LIN {X 0.130,Y -388.689,Z 418.603,A 0.000,B 0.000,C 90.000,E1 108.489} C_DIS
LIN {X -0.134,Y -405.495,Z 418.590,A 0.000,B 0.000,C 90.000,E1 106.260} C_DIS
LIN {X 0.180,Y -423.948,Z 418.578,A 0.000,B 0.000,C 90.000,E1 104.008} C_DIS
LIN {X -0.236,Y -443.839,Z 418.566,A 0.000,B 0.000,C 90.000,E1 101.951} C_DIS
LIN {X 0.157,Y -464.340,Z 418.555,A 0.000,B 0.000,C 90.000,E1 99.962} C_DIS
LIN {X -0.148,Y -485.345,Z 418.546,A 0.000,B 0.000,C 90.000,E1 98.219} C_DIS
LIN {X -0.012,Y -487.672,Z 418.544,A 0.000,B 0.000,C 90.000,E1 97.992} C_DIS
LIN {X 0.194,Y -489.436,Z 418.543,A 0.000,B 0.000,C 90.000,E1 97.757} C_DIS
LIN {X 0.023,Y -491.019,Z 418.542,A 0.000,B 0.000,C 90.000,E1 97.530} C_DIS
LIN {X -0.083,Y -492.202,Z 418.540,A 0.000,B 0.000,C 90.000,E1 97.296} C_DIS
LIN {X 0.146,Y -493.628,Z 418.538,A 0.000,B 0.000,C 90.000,E1 96.777} C_DIS
LIN {X -0.107,Y -494.007,Z 418.535,A 0.000,B 0.000,C 90.000,E1 96.315} C_DIS
LIN {X 0.138,Y -493.395,Z 418.532,A 0.000,B 0.000,C 90.000,E1 95.796} C_DIS
LIN {X -0.107,Y -491.696,Z 418.530,A 0.000,B 0.000,C 90.000,E1 95.334} C_DIS
LIN {X 0.236,Y -490.338,Z 418.528,A 0.000,B 0.000,C 90.000,E1 95.049} C_DIS
LIN {X -0.171,Y -484.764,Z 418.524,A 0.000,B 0.000,C 90.000,E1 94.359} C_DIS
LIN {X -0.157,Y -472.832,Z 418.516,A 0.000,B 0.000,C 90.000,E1 92.865} C_DIS
LIN {X -0.097,Y -455.462,Z 418.503,A 0.000,B 0.000,C 90.000,E1 90.573} C_DIS
LIN {X 0.061,Y -434.620,Z 418.486,A 0.000,B 0.000,C 90.000,E1 87.421} C_DIS
LIN {X 0.132,Y -413.786,Z 418.466,A 0.000,B 0.000,C 90.000,E1 83.913} C_DIS
LIN {X 0.008,Y -401.504,Z 418.454,A 0.000,B 0.000,C 90.000,E1 81.724} C_DIS
LIN {X 0.096,Y -390.851,Z 418.443,A 0.000,B 0.000,C 90.000,E1 79.746} C_DIS
LIN {X 0.073,Y -378.899,Z 418.430,A 0.000,B 0.000,C 90.000,E1 77.465} C_DIS
LIN {X -0.069,Y -365.997,Z 418.416,A 0.000,B 0.000,C 90.000,E1 74.866} C_DIS
LIN {X -0.041,Y -350.988,Z 418.398,A 0.000,B 0.000,C 90.000,E1 71.583} C_DIS
LIN {X -0.070,Y -338.219,Z 418.381,A 0.000,B 0.000,C 90.000,E1 68.539} C_DIS
LIN {X -0.050,Y -328.301,Z 418.367,A 0.000,B 0.000,C 90.000,E1 66.049} C_DIS
LIN {X 0.061,Y -319.808,Z 418.355,A 0.000,B 0.000,C 90.000,E1 63.819} C_DIS
LIN {X 0.144,Y -308.074,Z 418.337,A 0.000,B 0.000,C 90.000,E1 60.589} C_DIS
LIN {X 0.043,Y -297.005,Z 418.319,A 0.000,B 0.000,C 90.000,E1 57.327} C_DIS
LIN {X 0.032,Y -286.983,Z 418.300,A 0.000,B 0.000,C 90.000,E1 53.989} C_DIS
LIN {X 0.145,Y -279.385,Z 418.285,A 0.000,B 0.000,C 90.000,E1 51.251} C_DIS
LIN {X 0.000,Y -273.756,Z 418.273,A 0.000,B 0.000,C 90.000,E1 49.218} C_DIS
LIN {X -0.063,Y -267.896,Z 418.262,A 0.000,B 0.000,C 90.000,E1 47.148} C_DIS
LIN {X 0.124,Y -261.832,Z 418.250,A 0.000,B 0.000,C 90.000,E1 45.000} C_DIS
LIN {X 0.005,Y -255.633,Z 418.238,A 0.000,B 0.000,C 90.000,E1 42.894} C_DIS
LIN {X 0.002,Y -247.147,Z 418.222,A 0.000,B 0.000,C 90.000,E1 40.011} C_DIS
LIN {X -0.019,Y -236.856,Z 418.202,A 0.000,B 0.000,C 90.000,E1 36.343} C_DIS
LIN {X -0.108,Y -229.315,Z 418.185,A 0.000,B 0.000,C 90.000,E1 33.372} C_DIS
LIN {X -0.114,Y -222.425,Z 418.168,A 0.000,B 0.000,C 90.000,E1 30.335} C_DIS
LIN {X 0.062,Y -216.232,Z 418.151,A 0.000,B 0.000,C 90.000,E1 27.206} C_DIS
LIN {X -0.079,Y -209.441,Z 418.130,A 0.000,B 0.000,C 90.000,E1 23.334} C_DIS
LIN {X 0.087,Y -203.617,Z 418.107,A 0.000,B 0.000,C 90.000,E1 19.322} C_DIS
LIN {X 0.059,Y -198.758,Z 418.085,A 0.000,B 0.000,C 90.000,E1 15.315} C_DIS
LIN {X -0.095,Y -194.212,Z 418.058,A 0.000,B 0.000,C 90.000,E1 10.489} C_DIS
LIN {X -0.079,Y -191.040,Z 418.031,A 0.000,B 0.000,C 90.000,E1 5.568} C_DIS
LIN {X 0.073,Y -189.334,Z 417.993,A 0.000,B 0.000,C 90.000,E1 358.682} C_DIS
LIN {X -0.003,Y -191.373,Z 417.947,A 0.000,B 0.000,C 90.000,E1 350.443} C_DIS
LIN {X -0.026,Y -194.437,Z 417.919,A 0.000,B 0.000,C 90.000,E1 345.519} C_DIS
LIN {X -0.091,Y -198.077,Z 417.897,A 0.000,B 0.000,C 90.000,E1 341.456} C_DIS
LIN {X 0.089,Y -202.701,Z 417.874,A 0.000,B 0.000,C 90.000,E1 337.358} C_DIS
LIN {X -0.017,Y -208.427,Z 417.852,A 0.000,B 0.000,C 90.000,E1 333.384} C_DIS
LIN {X 0.026,Y -213.606,Z 417.835,A 0.000,B 0.000,C 90.000,E1 330.205} C_DIS
LIN {X 0.038,Y -220.600,Z 417.813,A 0.000,B 0.000,C 90.000,E1 326.294} C_DIS
LIN {X -0.092,Y -228.187,Z 417.791,A 0.000,B 0.000,C 90.000,E1 322.477} C_DIS
LIN {X -0.103,Y -236.777,Z 417.770,A 0.000,B 0.000,C 90.000,E1 318.690} C_DIS
LIN {X -0.037,Y -245.598,Z 417.752,A 0.000,B 0.000,C 90.000,E1 315.324} C_DIS
LIN {X 0.115,Y -254.400,Z 417.736,A 0.000,B 0.000,C 90.000,E1 312.366} C_DIS
LIN {X -0.143,Y -265.533,Z 417.718,A 0.000,B 0.000,C 90.000,E1 309.197} C_DIS
LIN {X 0.003,Y -277.655,Z 417.700,A 0.000,B 0.000,C 90.000,E1 306.011} C_DIS
LIN {X -0.128,Y -289.063,Z 417.685,A 0.000,B 0.000,C 90.000,E1 303.293} C_DIS
LIN {X -0.018,Y -303.956,Z 417.666,A 0.000,B 0.000,C 90.000,E1 299.922} C_DIS
LIN {X -0.031,Y -320.508,Z 417.648,A 0.000,B 0.000,C 90.000,E1 296.668} C_DIS
LIN {X -0.034,Y -335.095,Z 417.634,A 0.000,B 0.000,C 90.000,E1 294.131} C_DIS
LIN {X -0.001,Y -355.906,Z 417.617,A 0.000,B 0.000,C 90.000,E1 291.046} C_DIS
LIN {X 0.014,Y -376.407,Z 417.602,A 0.000,B 0.000,C 90.000,E1 288.362} C_DIS
LIN {X 0.077,Y -388.412,Z 417.594,A 0.000,B 0.000,C 90.000,E1 286.913} C_DIS
LIN {X 0.102,Y -403.817,Z 417.585,A 0.000,B 0.000,C 90.000,E1 285.245} C_DIS
LIN {X -0.137,Y -422.217,Z 417.575,A 0.000,B 0.000,C 90.000,E1 283.467} C_DIS
LIN {X 0.197,Y -432.492,Z 417.569,A 0.000,B 0.000,C 90.000,E1 282.411} C_DIS
LIN {X 0.001,Y -442.349,Z 417.563,A 0.000,B 0.000,C 90.000,E1 281.422} C_DIS
LIN {X -0.183,Y -449.356,Z 417.559,A 0.000,B 0.000,C 90.000,E1 280.658} C_DIS
LIN {X 0.023,Y -455.862,Z 417.555,A 0.000,B 0.000,C 90.000,E1 279.849} C_DIS
LIN {X 0.128,Y -463.718,Z 417.549,A 0.000,B 0.000,C 90.000,E1 278.803} C_DIS
LIN {X -0.141,Y -470.785,Z 417.543,A 0.000,B 0.000,C 90.000,E1 277.814} C_DIS
LIN {X -0.252,Y -475.616,Z 417.539,A 0.000,B 0.000,C 90.000,E1 277.068} C_DIS
LIN {X 0.210,Y -480.072,Z 417.535,A 0.000,B 0.000,C 90.000,E1 276.258} C_DIS
LIN {X 0.190,Y -484.015,Z 417.531,A 0.000,B 0.000,C 90.000,E1 275.511} C_DIS
LIN {X 0.243,Y -487.204,Z 417.527,A 0.000,B 0.000,C 90.000,E1 274.759} C_DIS
LIN {X -0.084,Y -488.885,Z 417.524,A 0.000,B 0.000,C 90.000,E1 274.302} C_DIS
LIN {X 0.119,Y -490.191,Z 417.521,A 0.000,B 0.000,C 90.000,E1 273.784} C_DIS
LIN {X -0.188,Y -491.163,Z 417.518,A 0.000,B 0.000,C 90.000,E1 273.326} C_DIS
LIN {X 0.030,Y -491.852,Z 417.516,A 0.000,B 0.000,C 90.000,E1 272.808} C_DIS
LIN {X 0.229,Y -492.166,Z 417.513,A 0.000,B 0.000,C 90.000,E1 272.293} C_DIS
LIN {X -0.058,Y -492.088,Z 417.510,A 0.000,B 0.000,C 90.000,E1 271.835} C_DIS
LIN {X 0.164,Y -491.562,Z 417.507,A 0.000,B 0.000,C 90.000,E1 271.318} C_DIS
LIN {X -0.120,Y -490.645,Z 417.505,A 0.000,B 0.000,C 90.000,E1 270.859} C_DIS
LIN {X 0.084,Y -489.178,Z 417.502,A 0.000,B 0.000,C 90.000,E1 270.344} C_DIS
LIN {X -0.205,Y -487.193,Z 417.499,A 0.000,B 0.000,C 90.000,E1 269.885} C_DIS
LIN {X -0.014,Y -484.575,Z 417.496,A 0.000,B 0.000,C 90.000,E1 269.370} C_DIS
LIN {X 0.154,Y -481.265,Z 417.494,A 0.000,B 0.000,C 90.000,E1 268.854} C_DIS
LIN {X -0.174,Y -477.014,Z 417.491,A 0.000,B 0.000,C 90.000,E1 268.396} C_DIS
LIN {X -0.030,Y -471.634,Z 417.488,A 0.000,B 0.000,C 90.000,E1 267.879} C_DIS
LIN {X -0.022,Y -468.790,Z 417.487,A 0.000,B 0.000,C 90.000,E1 267.650} C_DIS
LIN {X -0.013,Y -465.536,Z 417.486,A 0.000,B 0.000,C 90.000,E1 267.421} C_DIS
LIN {X -0.198,Y -462.346,Z 417.485,A 0.000,B 0.000,C 90.000,E1 267.249} C_DIS
LIN {X -0.238,Y -455.324,Z 417.483,A 0.000,B 0.000,C 90.000,E1 266.906} C_DIS
LIN {X -0.153,Y -448.247,Z 417.481,A 0.000,B 0.000,C 90.000,E1 266.617} C_DIS
LIN {X -0.141,Y -440.917,Z 417.480,A 0.000,B 0.000,C 90.000,E1 266.388} C_DIS
LIN {X -0.216,Y -433.025,Z 417.479,A 0.000,B 0.000,C 90.000,E1 266.216} C_DIS
LIN {X 0.047,Y -424.526,Z 417.478,A 0.000,B 0.000,C 90.000,E1 266.045} C_DIS
LIN {X 0.186,Y -412.102,Z 417.478,A 0.000,B 0.000,C 90.000,E1 265.931} C_DIS
LIN {X 0.148,Y -409.362,Z 417.477,A 0.000,B 0.000,C 90.000,E1 265.927} C_DIS
LIN {X 0.036,Y -180.917,Z 417.477,A 0.000,B 0.000,C 90.000,E1 265.927} C_DIS
LIN {X 0.040,Y -180.838,Z 417.472,A 0.000,B 0.000,C 90.000,E1 264.894} C_DIS
LIN {X -0.063,Y -178.878,Z 417.443,A 0.000,B 0.000,C 90.000,E1 259.690} C_DIS
LIN {X 0.013,Y -175.921,Z 417.414,A 0.000,B 0.000,C 90.000,E1 254.574} C_DIS
LIN {X -0.098,Y -174.618,Z 417.405,A 0.000,B 0.000,C 90.000,E1 252.906} C_DIS
LIN {X -0.005,Y -171.599,Z 417.381,A 0.000,B 0.000,C 90.000,E1 248.592} C_DIS
LIN {X -0.016,Y -167.821,Z 417.357,A 0.000,B 0.000,C 90.000,E1 244.280} C_DIS
LIN {X 0.001,Y -166.546,Z 417.347,A 0.000,B 0.000,C 90.000,E1 242.538} C_DIS
LIN {X -0.089,Y -162.542,Z 417.323,A 0.000,B 0.000,C 90.000,E1 238.201} C_DIS
LIN {X -0.028,Y -161.219,Z 417.313,A 0.000,B 0.000,C 90.000,E1 236.421} C_DIS
LIN {X 0.007,Y -157.226,Z 417.289,A 0.000,B 0.000,C 90.000,E1 231.984} C_DIS
LIN {X 0.031,Y -155.951,Z 417.279,A 0.000,B 0.000,C 90.000,E1 230.194} C_DIS
LIN {X -0.011,Y -152.205,Z 417.254,A 0.000,B 0.000,C 90.000,E1 225.729} C_DIS
LIN {X 0.011,Y -150.450,Z 417.239,A 0.000,B 0.000,C 90.000,E1 223.014} C_DIS
LIN {X 0.037,Y -147.176,Z 417.214,A 0.000,B 0.000,C 90.000,E1 218.463} C_DIS
LIN {X 0.004,Y -145.193,Z 417.193,A 0.000,B 0.000,C 90.000,E1 214.818} C_DIS
LIN {X 0.039,Y -142.333,Z 417.163,A 0.000,B 0.000,C 90.000,E1 209.283} C_DIS
LIN {X -0.032,Y -141.722,Z 417.152,A 0.000,B 0.000,C 90.000,E1 207.462} C_DIS
LIN {X -0.049,Y -139.478,Z 417.116,A 0.000,B 0.000,C 90.000,E1 200.972} C_DIS
LIN {X -0.061,Y -138.976,Z 417.101,A 0.000,B 0.000,C 90.000,E1 198.181} C_DIS
LIN {X 0.061,Y -138.331,Z 417.054,A 0.000,B 0.000,C 90.000,E1 189.726} C_DIS
LIN {X 0.064,Y -139.432,Z 417.007,A 0.000,B 0.000,C 90.000,E1 181.318} C_DIS
LIN {X 0.004,Y -140.959,Z 416.976,A 0.000,B 0.000,C 90.000,E1 175.755} C_DIS
LIN {X -0.046,Y -142.715,Z 416.956,A 0.000,B 0.000,C 90.000,E1 172.064} C_DIS
LIN {X 0.054,Y -145.094,Z 416.930,A 0.000,B 0.000,C 90.000,E1 167.409} C_DIS
LIN {X 0.049,Y -147.718,Z 416.910,A 0.000,B 0.000,C 90.000,E1 163.740} C_DIS
LIN {X -0.010,Y -150.375,Z 416.889,A 0.000,B 0.000,C 90.000,E1 160.115} C_DIS
LIN {X 0.008,Y -153.805,Z 416.869,A 0.000,B 0.000,C 90.000,E1 156.485} C_DIS
LIN {X 0.068,Y -157.216,Z 416.849,A 0.000,B 0.000,C 90.000,E1 152.871} C_DIS
LIN {X 0.008,Y -161.381,Z 416.830,A 0.000,B 0.000,C 90.000,E1 149.331} C_DIS
LIN {X 0.020,Y -165.583,Z 416.810,A 0.000,B 0.000,C 90.000,E1 145.801} C_DIS
LIN {X 0.006,Y -170.506,Z 416.791,A 0.000,B 0.000,C 90.000,E1 142.316} C_DIS
LIN {X 0.050,Y -175.385,Z 416.771,A 0.000,B 0.000,C 90.000,E1 138.852} C_DIS
LIN {X -0.087,Y -181.009,Z 416.753,A 0.000,B 0.000,C 90.000,E1 135.486} C_DIS
LIN {X 0.037,Y -186.439,Z 416.734,A 0.000,B 0.000,C 90.000,E1 132.081} C_DIS
LIN {X 0.106,Y -191.064,Z 416.720,A 0.000,B 0.000,C 90.000,E1 129.564} C_DIS
LIN {X -0.035,Y -196.732,Z 416.702,A 0.000,B 0.000,C 90.000,E1 126.377} C_DIS
LIN {X -0.087,Y -294.757,Z 416.702,A 0.000,B 0.000,C 90.000,E1 126.377} C_DIS
LIN {X 0.042,Y -297.998,Z 416.702,A 0.000,B 0.000,C 90.000,E1 126.297} C_DIS
LIN {X 0.063,Y -300.668,Z 416.701,A 0.000,B 0.000,C 90.000,E1 126.171} C_DIS
LIN {X 0.071,Y -304.249,Z 416.699,A 0.000,B 0.000,C 90.000,E1 125.884} C_DIS
LIN {X -0.057,Y -307.884,Z 416.697,A 0.000,B 0.000,C 90.000,E1 125.438} C_DIS
LIN {X -0.031,Y -309.677,Z 416.695,A 0.000,B 0.000,C 90.000,E1 125.105} C_DIS
LIN {X -0.004,Y -311.083,Z 416.693,A 0.000,B 0.000,C 90.000,E1 124.771} C_DIS
LIN {X 0.092,Y -323.167,Z 416.673,A 0.000,B 0.000,C 90.000,E1 121.209} C_DIS
LIN {X 0.136,Y -334.446,Z 416.658,A 0.000,B 0.000,C 90.000,E1 118.359} C_DIS
LIN {X 0.024,Y -347.149,Z 416.642,A 0.000,B 0.000,C 90.000,E1 115.591} C_DIS
LIN {X 0.094,Y -359.734,Z 416.629,A 0.000,B 0.000,C 90.000,E1 113.153} C_DIS
LIN {X 0.010,Y -373.629,Z 416.616,A 0.000,B 0.000,C 90.000,E1 110.791} C_DIS
LIN {X -0.133,Y -388.936,Z 416.603,A 0.000,B 0.000,C 90.000,E1 108.489} C_DIS
LIN {X -0.013,Y -405.767,Z 416.590,A 0.000,B 0.000,C 90.000,E1 106.205} C_DIS
LIN {X -0.093,Y -424.249,Z 416.578,A 0.000,B 0.000,C 90.000,E1 104.008} C_DIS
LIN {X 0.024,Y -444.153,Z 416.566,A 0.000,B 0.000,C 90.000,E1 101.883} C_DIS
LIN {X -0.099,Y -464.664,Z 416.555,A 0.000,B 0.000,C 90.000,E1 99.962} C_DIS
LIN {X 0.086,Y -485.676,Z 416.545,A 0.000,B 0.000,C 90.000,E1 98.163} C_DIS
LIN {X 0.207,Y -487.985,Z 416.544,A 0.000,B 0.000,C 90.000,E1 97.936} C_DIS
LIN {X 0.231,Y -489.872,Z 416.543,A 0.000,B 0.000,C 90.000,E1 97.701} C_DIS
LIN {X 0.190,Y -491.309,Z 416.542,A 0.000,B 0.000,C 90.000,E1 97.473} C_DIS
LIN {X -0.013,Y -493.295,Z 416.539,A 0.000,B 0.000,C 90.000,E1 97.004} C_DIS
LIN {X 0.217,Y -494.139,Z 416.536,A 0.000,B 0.000,C 90.000,E1 96.486} C_DIS
LIN {X -0.084,Y -493.986,Z 416.533,A 0.000,B 0.000,C 90.000,E1 96.030} C_DIS
LIN {X 0.166,Y -492.812,Z 416.531,A 0.000,B 0.000,C 90.000,E1 95.511} C_DIS
LIN {X 0.067,Y -491.785,Z 416.529,A 0.000,B 0.000,C 90.000,E1 95.277} C_DIS
LIN {X -0.077,Y -490.395,Z 416.528,A 0.000,B 0.000,C 90.000,E1 95.049} C_DIS
LIN {X -0.155,Y -482.849,Z 416.523,A 0.000,B 0.000,C 90.000,E1 94.073} C_DIS
LIN {X -0.172,Y -470.860,Z 416.514,A 0.000,B 0.000,C 90.000,E1 92.579} C_DIS
LIN {X -0.157,Y -453.666,Z 416.501,A 0.000,B 0.000,C 90.000,E1 90.286} C_DIS
LIN {X 0.095,Y -431.317,Z 416.483,A 0.000,B 0.000,C 90.000,E1 86.849} C_DIS
LIN {X 0.068,Y -410.717,Z 416.463,A 0.000,B 0.000,C 90.000,E1 83.337} C_DIS
LIN {X -0.157,Y -399.969,Z 416.452,A 0.000,B 0.000,C 90.000,E1 81.432} C_DIS
LIN {X -0.092,Y -389.369,Z 416.441,A 0.000,B 0.000,C 90.000,E1 79.454} C_DIS
LIN {X -0.146,Y -377.488,Z 416.429,A 0.000,B 0.000,C 90.000,E1 77.173} C_DIS
LIN {X 0.050,Y -366.026,Z 416.416,A 0.000,B 0.000,C 90.000,E1 74.810} C_DIS
LIN {X 0.140,Y -352.300,Z 416.399,A 0.000,B 0.000,C 90.000,E1 71.819} C_DIS
LIN {X 0.146,Y -340.701,Z 416.384,A 0.000,B 0.000,C 90.000,E1 69.082} C_DIS
LIN {X 0.096,Y -330.713,Z 416.370,A 0.000,B 0.000,C 90.000,E1 66.613} C_DIS
LIN {X 0.060,Y -320.929,Z 416.356,A 0.000,B 0.000,C 90.000,E1 64.101} C_DIS
LIN {X -0.107,Y -309.129,Z 416.338,A 0.000,B 0.000,C 90.000,E1 60.923} C_DIS
LIN {X -0.167,Y -297.962,Z 416.320,A 0.000,B 0.000,C 90.000,E1 57.661} C_DIS
LIN {X 0.096,Y -287.853,Z 416.302,A 0.000,B 0.000,C 90.000,E1 54.276} C_DIS
LIN {X -0.165,Y -280.242,Z 416.287,A 0.000,B 0.000,C 90.000,E1 51.618} C_DIS
LIN {X -0.079,Y -274.614,Z 416.275,A 0.000,B 0.000,C 90.000,E1 49.542} C_DIS
LIN {X -0.128,Y -268.837,Z 416.264,A 0.000,B 0.000,C 90.000,E1 47.472} C_DIS
LIN {X 0.077,Y -262.787,Z 416.252,A 0.000,B 0.000,C 90.000,E1 45.324} C_DIS
LIN {X -0.022,Y -256.648,Z 416.240,A 0.000,B 0.000,C 90.000,E1 43.218} C_DIS
LIN {X 0.005,Y -248.174,Z 416.224,A 0.000,B 0.000,C 90.000,E1 40.334} C_DIS
LIN {X 0.049,Y -239.893,Z 416.208,A 0.000,B 0.000,C 90.000,E1 37.397} C_DIS
LIN {X 0.115,Y -232.068,Z 416.191,A 0.000,B 0.000,C 90.000,E1 34.405} C_DIS
LIN {X -0.019,Y -224.954,Z 416.174,A 0.000,B 0.000,C 90.000,E1 31.416} C_DIS
LIN {X -0.056,Y -218.476,Z 416.157,A 0.000,B 0.000,C 90.000,E1 28.359} C_DIS
LIN {X -0.038,Y -211.378,Z 416.136,A 0.000,B 0.000,C 90.000,E1 24.463} C_DIS
LIN {X 0.074,Y -205.249,Z 416.114,A 0.000,B 0.000,C 90.000,E1 20.482} C_DIS
LIN {X 0.020,Y -200.060,Z 416.092,A 0.000,B 0.000,C 90.000,E1 16.496} C_DIS
LIN {X -0.074,Y -195.889,Z 416.069,A 0.000,B 0.000,C 90.000,E1 12.479} C_DIS
LIN {X -0.102,Y -192.079,Z 416.042,A 0.000,B 0.000,C 90.000,E1 7.587} C_DIS
LIN {X -0.022,Y -189.422,Z 416.005,A 0.000,B 0.000,C 90.000,E1 0.974} C_DIS
LIN {X 0.038,Y -190.876,Z 415.951,A 0.000,B 0.000,C 90.000,E1 351.254} C_DIS
LIN {X -0.037,Y -194.307,Z 415.919,A 0.000,B 0.000,C 90.000,E1 345.519} C_DIS
LIN {X 0.082,Y -197.950,Z 415.897,A 0.000,B 0.000,C 90.000,E1 341.402} C_DIS
LIN {X 0.068,Y -202.554,Z 415.874,A 0.000,B 0.000,C 90.000,E1 337.358} C_DIS
LIN {X -0.042,Y -208.273,Z 415.852,A 0.000,B 0.000,C 90.000,E1 333.384} C_DIS
LIN {X 0.031,Y -214.780,Z 415.830,A 0.000,B 0.000,C 90.000,E1 329.410} C_DIS
LIN {X 0.002,Y -220.476,Z 415.813,A 0.000,B 0.000,C 90.000,E1 326.294} C_DIS
LIN {X 0.047,Y -228.082,Z 415.791,A 0.000,B 0.000,C 90.000,E1 322.431} C_DIS
LIN {X 0.029,Y -236.679,Z 415.770,A 0.000,B 0.000,C 90.000,E1 318.647} C_DIS
LIN {X -0.088,Y -245.509,Z 415.752,A 0.000,B 0.000,C 90.000,E1 315.324} C_DIS
LIN {X -0.128,Y -253.143,Z 415.737,A 0.000,B 0.000,C 90.000,E1 312.771} C_DIS
LIN {X 0.118,Y -264.176,Z 415.719,A 0.000,B 0.000,C 90.000,E1 309.483} C_DIS
LIN {X -0.158,Y -276.215,Z 415.702,A 0.000,B 0.000,C 90.000,E1 306.377} C_DIS
LIN {X 0.044,Y -288.999,Z 415.685,A 0.000,B 0.000,C 90.000,E1 303.245} C_DIS
LIN {X -0.094,Y -303.874,Z 415.666,A 0.000,B 0.000,C 90.000,E1 299.922} C_DIS
LIN {X 0.174,Y -320.475,Z 415.648,A 0.000,B 0.000,C 90.000,E1 296.616} C_DIS
LIN {X -0.119,Y -335.147,Z 415.634,A 0.000,B 0.000,C 90.000,E1 294.131} C_DIS
LIN {X -0.126,Y -353.840,Z 415.619,A 0.000,B 0.000,C 90.000,E1 291.354} C_DIS
LIN {X -0.076,Y -376.529,Z 415.602,A 0.000,B 0.000,C 90.000,E1 288.362} C_DIS
LIN {X -0.184,Y -386.139,Z 415.596,A 0.000,B 0.000,C 90.000,E1 287.221} C_DIS
LIN {X 0.130,Y -403.898,Z 415.585,A 0.000,B 0.000,C 90.000,E1 285.245} C_DIS
LIN {X -0.074,Y -422.208,Z 415.575,A 0.000,B 0.000,C 90.000,E1 283.467} C_DIS
LIN {X 0.249,Y -432.518,Z 415.569,A 0.000,B 0.000,C 90.000,E1 282.411} C_DIS
LIN {X -0.228,Y -439.953,Z 415.565,A 0.000,B 0.000,C 90.000,E1 281.715} C_DIS
LIN {X 0.121,Y -447.068,Z 415.561,A 0.000,B 0.000,C 90.000,E1 280.894} C_DIS
LIN {X -0.129,Y -453.708,Z 415.556,A 0.000,B 0.000,C 90.000,E1 280.141} C_DIS
LIN {X -0.052,Y -461.750,Z 415.550,A 0.000,B 0.000,C 90.000,E1 279.095} C_DIS
LIN {X 0.122,Y -469.024,Z 415.545,A 0.000,B 0.000,C 90.000,E1 278.049} C_DIS
LIN {X -0.152,Y -475.552,Z 415.539,A 0.000,B 0.000,C 90.000,E1 277.068} C_DIS
LIN {X 0.124,Y -481.402,Z 415.534,A 0.000,B 0.000,C 90.000,E1 276.030} C_DIS
LIN {X 0.158,Y -485.052,Z 415.529,A 0.000,B 0.000,C 90.000,E1 275.277} C_DIS
LIN {X -0.183,Y -487.102,Z 415.527,A 0.000,B 0.000,C 90.000,E1 274.821} C_DIS
LIN {X 0.017,Y -488.814,Z 415.524,A 0.000,B 0.000,C 90.000,E1 274.302} C_DIS
LIN {X 0.220,Y -490.131,Z 415.521,A 0.000,B 0.000,C 90.000,E1 273.784} C_DIS
LIN {X -0.088,Y -491.131,Z 415.518,A 0.000,B 0.000,C 90.000,E1 273.326} C_DIS
LIN {X 0.130,Y -491.784,Z 415.516,A 0.000,B 0.000,C 90.000,E1 272.808} C_DIS
LIN {X -0.164,Y -492.126,Z 415.513,A 0.000,B 0.000,C 90.000,E1 272.350} C_DIS
LIN {X 0.042,Y -492.033,Z 415.510,A 0.000,B 0.000,C 90.000,E1 271.835} C_DIS
LIN {X -0.228,Y -491.549,Z 415.507,A 0.000,B 0.000,C 90.000,E1 271.375} C_DIS
LIN {X -0.022,Y -490.623,Z 415.505,A 0.000,B 0.000,C 90.000,E1 270.859} C_DIS
LIN {X 0.183,Y -489.221,Z 415.502,A 0.000,B 0.000,C 90.000,E1 270.344} C_DIS
LIN {X -0.106,Y -487.265,Z 415.499,A 0.000,B 0.000,C 90.000,E1 269.885} C_DIS
LIN {X 0.083,Y -484.707,Z 415.497,A 0.000,B 0.000,C 90.000,E1 269.370} C_DIS
LIN {X -0.229,Y -481.382,Z 415.494,A 0.000,B 0.000,C 90.000,E1 268.912} C_DIS
LIN {X 0.088,Y -479.409,Z 415.492,A 0.000,B 0.000,C 90.000,E1 268.625} C_DIS
LIN {X 0.240,Y -474.679,Z 415.490,A 0.000,B 0.000,C 90.000,E1 268.108} C_DIS
LIN {X 0.067,Y -471.871,Z 415.488,A 0.000,B 0.000,C 90.000,E1 267.879} C_DIS
LIN {X 0.061,Y -465.731,Z 415.486,A 0.000,B 0.000,C 90.000,E1 267.421} C_DIS
LIN {X -0.140,Y -462.531,Z 415.485,A 0.000,B 0.000,C 90.000,E1 267.249} C_DIS
LIN {X -0.192,Y -455.516,Z 415.483,A 0.000,B 0.000,C 90.000,E1 266.906} C_DIS
LIN {X -0.108,Y -448.412,Z 415.481,A 0.000,B 0.000,C 90.000,E1 266.617} C_DIS
LIN {X -0.120,Y -441.189,Z 415.480,A 0.000,B 0.000,C 90.000,E1 266.388} C_DIS
LIN {X -0.216,Y -433.199,Z 415.479,A 0.000,B 0.000,C 90.000,E1 266.216} C_DIS
LIN {X 0.050,Y -424.671,Z 415.478,A 0.000,B 0.000,C 90.000,E1 266.045} C_DIS
LIN {X -0.085,Y -415.957,Z 415.478,A 0.000,B 0.000,C 90.000,E1 265.988} C_DIS
LIN {X 0.150,Y -409.759,Z 415.477,A 0.000,B 0.000,C 90.000,E1 265.927} C_DIS
LIN {X 0.036,Y -180.917,Z 415.477,A 0.000,B 0.000,C 90.000,E1 265.927} C_DIS
LIN {X 0.039,Y -180.838,Z 415.472,A 0.000,B 0.000,C 90.000,E1 264.894} C_DIS
LIN {X -0.064,Y -178.879,Z 415.443,A 0.000,B 0.000,C 90.000,E1 259.690} C_DIS
LIN {X 0.012,Y -175.921,Z 415.414,A 0.000,B 0.000,C 90.000,E1 254.574} C_DIS
LIN {X -0.098,Y -174.618,Z 415.405,A 0.000,B 0.000,C 90.000,E1 252.906} C_DIS
LIN {X -0.005,Y -171.599,Z 415.381,A 0.000,B 0.000,C 90.000,E1 248.592} C_DIS
LIN {X -0.017,Y -167.822,Z 415.357,A 0.000,B 0.000,C 90.000,E1 244.280} C_DIS
LIN {X 0.001,Y -166.545,Z 415.347,A 0.000,B 0.000,C 90.000,E1 242.538} C_DIS
LIN {X -0.089,Y -162.542,Z 415.323,A 0.000,B 0.000,C 90.000,E1 238.201} C_DIS
LIN {X -0.029,Y -161.218,Z 415.313,A 0.000,B 0.000,C 90.000,E1 236.421} C_DIS
LIN {X 0.007,Y -157.225,Z 415.289,A 0.000,B 0.000,C 90.000,E1 231.984} C_DIS
LIN {X 0.029,Y -155.951,Z 415.279,A 0.000,B 0.000,C 90.000,E1 230.194} C_DIS
LIN {X -0.011,Y -152.204,Z 415.254,A 0.000,B 0.000,C 90.000,E1 225.729} C_DIS
LIN {X 0.010,Y -150.449,Z 415.239,A 0.000,B 0.000,C 90.000,E1 223.014} C_DIS
LIN {X 0.037,Y -147.175,Z 415.214,A 0.000,B 0.000,C 90.000,E1 218.463} C_DIS
LIN {X 0.003,Y -145.192,Z 415.193,A 0.000,B 0.000,C 90.000,E1 214.818} C_DIS
LIN {X 0.038,Y -142.333,Z 415.163,A 0.000,B 0.000,C 90.000,E1 209.283} C_DIS
LIN {X -0.033,Y -141.722,Z 415.152,A 0.000,B 0.000,C 90.000,E1 207.462} C_DIS
LIN {X -0.050,Y -139.477,Z 415.116,A 0.000,B 0.000,C 90.000,E1 200.972} C_DIS
LIN {X -0.062,Y -138.975,Z 415.101,A 0.000,B 0.000,C 90.000,E1 198.181} C_DIS
LIN {X 0.060,Y -138.331,Z 415.054,A 0.000,B 0.000,C 90.000,E1 189.726} C_DIS
LIN {X 0.063,Y -139.432,Z 415.007,A 0.000,B 0.000,C 90.000,E1 181.318} C_DIS
LIN {X 0.003,Y -140.959,Z 414.976,A 0.000,B 0.000,C 90.000,E1 175.755} C_DIS
LIN {X -0.047,Y -142.715,Z 414.956,A 0.000,B 0.000,C 90.000,E1 172.064} C_DIS
LIN {X 0.053,Y -145.094,Z 414.930,A 0.000,B 0.000,C 90.000,E1 167.409} C_DIS
LIN {X 0.048,Y -147.718,Z 414.910,A 0.000,B 0.000,C 90.000,E1 163.740} C_DIS
LIN {X -0.010,Y -150.376,Z 414.889,A 0.000,B 0.000,C 90.000,E1 160.115} C_DIS
LIN {X 0.007,Y -153.804,Z 414.869,A 0.000,B 0.000,C 90.000,E1 156.485} C_DIS
LIN {X 0.067,Y -157.217,Z 414.849,A 0.000,B 0.000,C 90.000,E1 152.871} C_DIS
LIN {X 0.008,Y -161.381,Z 414.830,A 0.000,B 0.000,C 90.000,E1 149.331} C_DIS
LIN {X 0.019,Y -165.584,Z 414.810,A 0.000,B 0.000,C 90.000,E1 145.801} C_DIS
LIN {X 0.005,Y -170.505,Z 414.791,A 0.000,B 0.000,C 90.000,E1 142.316} C_DIS
LIN {X 0.050,Y -175.386,Z 414.771,A 0.000,B 0.000,C 90.000,E1 138.852} C_DIS
LIN {X -0.088,Y -181.010,Z 414.753,A 0.000,B 0.000,C 90.000,E1 135.486} C_DIS
LIN {X 0.036,Y -186.439,Z 414.734,A 0.000,B 0.000,C 90.000,E1 132.081} C_DIS
LIN {X 0.105,Y -191.064,Z 414.720,A 0.000,B 0.000,C 90.000,E1 129.564} C_DIS
LIN {X 0.065,Y -196.830,Z 414.702,A 0.000,B 0.000,C 90.000,E1 126.297} C_DIS
LIN {X 0.041,Y -294.947,Z 414.702,A 0.000,B 0.000,C 90.000,E1 126.297} C_DIS
LIN {X -0.034,Y -299.200,Z 414.701,A 0.000,B 0.000,C 90.000,E1 126.217} C_DIS
LIN {X 0.093,Y -302.292,Z 414.700,A 0.000,B 0.000,C 90.000,E1 126.011} C_DIS
LIN {X -0.051,Y -305.950,Z 414.698,A 0.000,B 0.000,C 90.000,E1 125.678} C_DIS
LIN {X 0.029,Y -309.503,Z 414.695,A 0.000,B 0.000,C 90.000,E1 125.105} C_DIS
LIN {X 0.060,Y -310.975,Z 414.693,A 0.000,B 0.000,C 90.000,E1 124.771} C_DIS
LIN {X 0.035,Y -317.426,Z 414.682,A 0.000,B 0.000,C 90.000,E1 122.832} C_DIS
LIN {X 0.080,Y -327.951,Z 414.666,A 0.000,B 0.000,C 90.000,E1 119.951} C_DIS
LIN {X 0.103,Y -339.843,Z 414.651,A 0.000,B 0.000,C 90.000,E1 117.129} C_DIS
LIN {X -0.016,Y -353.214,Z 414.635,A 0.000,B 0.000,C 90.000,E1 114.387} C_DIS
LIN {X 0.068,Y -366.438,Z 414.622,A 0.000,B 0.000,C 90.000,E1 111.972} C_DIS
LIN {X 0.010,Y -381.020,Z 414.609,A 0.000,B 0.000,C 90.000,E1 109.631} C_DIS
LIN {X 0.048,Y -397.070,Z 414.596,A 0.000,B 0.000,C 90.000,E1 107.330} C_DIS
LIN {X 0.148,Y -414.704,Z 414.584,A 0.000,B 0.000,C 90.000,E1 105.079} C_DIS
LIN {X -0.095,Y -434.015,Z 414.572,A 0.000,B 0.000,C 90.000,E1 102.939} C_DIS
LIN {X 0.067,Y -454.247,Z 414.561,A 0.000,B 0.000,C 90.000,E1 100.894} C_DIS
LIN {X 0.152,Y -475.016,Z 414.550,A 0.000,B 0.000,C 90.000,E1 99.029} C_DIS
LIN {X 0.130,Y -485.580,Z 414.545,A 0.000,B 0.000,C 90.000,E1 98.163} C_DIS
LIN {X -0.214,Y -487.936,Z 414.544,A 0.000,B 0.000,C 90.000,E1 97.992} C_DIS
LIN {X -0.007,Y -489.724,Z 414.543,A 0.000,B 0.000,C 90.000,E1 97.757} C_DIS
LIN {X -0.178,Y -491.327,Z 414.542,A 0.000,B 0.000,C 90.000,E1 97.530} C_DIS
LIN {X 0.204,Y -492.527,Z 414.540,A 0.000,B 0.000,C 90.000,E1 97.239} C_DIS
LIN {X -0.053,Y -493.980,Z 414.538,A 0.000,B 0.000,C 90.000,E1 96.777} C_DIS
LIN {X 0.187,Y -494.381,Z 414.535,A 0.000,B 0.000,C 90.000,E1 96.258} C_DIS
LIN {X -0.057,Y -493.793,Z 414.532,A 0.000,B 0.000,C 90.000,E1 95.796} C_DIS
LIN {X 0.191,Y -492.119,Z 414.529,A 0.000,B 0.000,C 90.000,E1 95.277} C_DIS
LIN {X 0.046,Y -490.777,Z 414.528,A 0.000,B 0.000,C 90.000,E1 95.049} C_DIS
LIN {X -0.030,Y -483.303,Z 414.523,A 0.000,B 0.000,C 90.000,E1 94.073} C_DIS
LIN {X -0.042,Y -471.314,Z 414.514,A 0.000,B 0.000,C 90.000,E1 92.579} C_DIS
LIN {X -0.015,Y -454.090,Z 414.502,A 0.000,B 0.000,C 90.000,E1 90.286} C_DIS
LIN {X -0.190,Y -431.668,Z 414.483,A 0.000,B 0.000,C 90.000,E1 86.906} C_DIS
LIN {X -0.185,Y -411.063,Z 414.463,A 0.000,B 0.000,C 90.000,E1 83.394} C_DIS
LIN {X 0.087,Y -398.777,Z 414.451,A 0.000,B 0.000,C 90.000,E1 81.141} C_DIS
LIN {X 0.178,Y -386.729,Z 414.438,A 0.000,B 0.000,C 90.000,E1 78.870} C_DIS
LIN {X 0.154,Y -372.084,Z 414.422,A 0.000,B 0.000,C 90.000,E1 75.992} C_DIS
LIN {X -0.122,Y -358.011,Z 414.406,A 0.000,B 0.000,C 90.000,E1 73.087} C_DIS
LIN {X -0.034,Y -343.492,Z 414.387,A 0.000,B 0.000,C 90.000,E1 69.752} C_DIS
LIN {X -0.018,Y -332.165,Z 414.372,A 0.000,B 0.000,C 90.000,E1 66.975} C_DIS
LIN {X -0.006,Y -322.300,Z 414.358,A 0.000,B 0.000,C 90.000,E1 64.460} C_DIS
LIN {X 0.008,Y -310.418,Z 414.340,A 0.000,B 0.000,C 90.000,E1 61.257} C_DIS
LIN {X -0.020,Y -299.180,Z 414.322,A 0.000,B 0.000,C 90.000,E1 57.995} C_DIS
LIN {X -0.128,Y -288.933,Z 414.304,A 0.000,B 0.000,C 90.000,E1 54.689} C_DIS
LIN {X -0.131,Y -281.277,Z 414.289,A 0.000,B 0.000,C 90.000,E1 51.984} C_DIS
LIN {X -0.026,Y -275.675,Z 414.277,A 0.000,B 0.000,C 90.000,E1 49.908} C_DIS
LIN {X -0.054,Y -269.948,Z 414.266,A 0.000,B 0.000,C 90.000,E1 47.838} C_DIS
LIN {X -0.009,Y -263.961,Z 414.254,A 0.000,B 0.000,C 90.000,E1 45.729} C_DIS
LIN {X -0.084,Y -257.852,Z 414.242,A 0.000,B 0.000,C 90.000,E1 43.623} C_DIS
LIN {X -0.048,Y -249.439,Z 414.226,A 0.000,B 0.000,C 90.000,E1 40.744} C_DIS
LIN {X 0.019,Y -241.167,Z 414.210,A 0.000,B 0.000,C 90.000,E1 37.810} C_DIS
LIN {X 0.115,Y -233.222,Z 414.194,A 0.000,B 0.000,C 90.000,E1 34.818} C_DIS
LIN {X 0.071,Y -224.329,Z 414.173,A 0.000,B 0.000,C 90.000,E1 31.052} C_DIS
LIN {X 0.093,Y -217.902,Z 414.156,A 0.000,B 0.000,C 90.000,E1 27.975} C_DIS
LIN {X -0.045,Y -212.183,Z 414.138,A 0.000,B 0.000,C 90.000,E1 24.899} C_DIS
LIN {X 0.094,Y -205.914,Z 414.116,A 0.000,B 0.000,C 90.000,E1 20.918} C_DIS
LIN {X -0.067,Y -200.580,Z 414.094,A 0.000,B 0.000,C 90.000,E1 16.968} C_DIS
LIN {X 0.087,Y -196.272,Z 414.072,A 0.000,B 0.000,C 90.000,E1 12.883} C_DIS
LIN {X 0.066,Y -192.295,Z 414.045,A 0.000,B 0.000,C 90.000,E1 7.992} C_DIS
LIN {X 0.049,Y -189.627,Z 414.013,A 0.000,B 0.000,C 90.000,E1 2.236} C_DIS
LIN {X 0.032,Y -190.763,Z 413.951,A 0.000,B 0.000,C 90.000,E1 351.254} C_DIS
LIN {X -0.093,Y -193.581,Z 413.924,A 0.000,B 0.000,C 90.000,E1 346.353} C_DIS
LIN {X -0.001,Y -196.986,Z 413.901,A 0.000,B 0.000,C 90.000,E1 342.236} C_DIS
LIN {X 0.079,Y -201.377,Z 413.879,A 0.000,B 0.000,C 90.000,E1 338.156} C_DIS
LIN {X 0.037,Y -206.882,Z 413.856,A 0.000,B 0.000,C 90.000,E1 334.152} C_DIS
LIN {X -0.034,Y -213.274,Z 413.834,A 0.000,B 0.000,C 90.000,E1 330.205} C_DIS
LIN {X -0.035,Y -220.361,Z 413.813,A 0.000,B 0.000,C 90.000,E1 326.294} C_DIS
LIN {X 0.006,Y -227.983,Z 413.791,A 0.000,B 0.000,C 90.000,E1 322.431} C_DIS
LIN {X 0.063,Y -234.773,Z 413.774,A 0.000,B 0.000,C 90.000,E1 319.380} C_DIS
LIN {X 0.101,Y -242.382,Z 413.758,A 0.000,B 0.000,C 90.000,E1 316.377} C_DIS
LIN {X -0.006,Y -251.893,Z 413.739,A 0.000,B 0.000,C 90.000,E1 313.095} C_DIS
LIN {X 0.008,Y -262.806,Z 413.721,A 0.000,B 0.000,C 90.000,E1 309.850} C_DIS
LIN {X -0.011,Y -273.415,Z 413.706,A 0.000,B 0.000,C 90.000,E1 307.030} C_DIS
LIN {X 0.041,Y -286.041,Z 413.688,A 0.000,B 0.000,C 90.000,E1 303.913} C_DIS
LIN {X 0.054,Y -297.666,Z 413.673,A 0.000,B 0.000,C 90.000,E1 301.209} C_DIS
LIN {X 0.063,Y -310.239,Z 413.659,A 0.000,B 0.000,C 90.000,E1 298.565} C_DIS
LIN {X 0.097,Y -324.025,Z 413.644,A 0.000,B 0.000,C 90.000,E1 295.976} C_DIS
LIN {X 0.074,Y -337.185,Z 413.632,A 0.000,B 0.000,C 90.000,E1 293.770} C_DIS
LIN {X -0.142,Y -358.349,Z 413.615,A 0.000,B 0.000,C 90.000,E1 290.737} C_DIS
LIN {X -0.165,Y -376.656,Z 413.602,A 0.000,B 0.000,C 90.000,E1 288.362} C_DIS
LIN {X 0.058,Y -386.366,Z 413.595,A 0.000,B 0.000,C 90.000,E1 287.166} C_DIS
LIN {X 0.030,Y -404.156,Z 413.585,A 0.000,B 0.000,C 90.000,E1 285.245} C_DIS
LIN {X -0.149,Y -422.407,Z 413.575,A 0.000,B 0.000,C 90.000,E1 283.467} C_DIS
LIN {X 0.034,Y -435.124,Z 413.568,A 0.000,B 0.000,C 90.000,E1 282.187} C_DIS
LIN {X -0.021,Y -442.544,Z 413.563,A 0.000,B 0.000,C 90.000,E1 281.422} C_DIS
LIN {X 0.232,Y -449.558,Z 413.559,A 0.000,B 0.000,C 90.000,E1 280.602} C_DIS
LIN {X -0.002,Y -455.979,Z 413.555,A 0.000,B 0.000,C 90.000,E1 279.849} C_DIS
LIN {X 0.104,Y -463.774,Z 413.549,A 0.000,B 0.000,C 90.000,E1 278.803} C_DIS
LIN {X -0.165,Y -470.828,Z 413.543,A 0.000,B 0.000,C 90.000,E1 277.814} C_DIS
LIN {X 0.049,Y -477.187,Z 413.538,A 0.000,B 0.000,C 90.000,E1 276.777} C_DIS
LIN {X -0.001,Y -481.455,Z 413.534,A 0.000,B 0.000,C 90.000,E1 276.030} C_DIS
LIN {X 0.034,Y -485.122,Z 413.529,A 0.000,B 0.000,C 90.000,E1 275.277} C_DIS
LIN {X 0.218,Y -487.169,Z 413.527,A 0.000,B 0.000,C 90.000,E1 274.759} C_DIS
LIN {X -0.109,Y -488.824,Z 413.524,A 0.000,B 0.000,C 90.000,E1 274.302} C_DIS
LIN {X 0.095,Y -490.156,Z 413.521,A 0.000,B 0.000,C 90.000,E1 273.784} C_DIS
LIN {X -0.214,Y -491.112,Z 413.518,A 0.000,B 0.000,C 90.000,E1 273.326} C_DIS
LIN {X 0.004,Y -491.744,Z 413.516,A 0.000,B 0.000,C 90.000,E1 272.808} C_DIS
LIN {X 0.203,Y -492.061,Z 413.513,A 0.000,B 0.000,C 90.000,E1 272.293} C_DIS
LIN {X -0.084,Y -491.994,Z 413.510,A 0.000,B 0.000,C 90.000,E1 271.835} C_DIS
LIN {X 0.137,Y -491.502,Z 413.507,A 0.000,B 0.000,C 90.000,E1 271.318} C_DIS
LIN {X -0.147,Y -490.485,Z 413.505,A 0.000,B 0.000,C 90.000,E1 270.859} C_DIS
LIN {X 0.057,Y -489.169,Z 413.502,A 0.000,B 0.000,C 90.000,E1 270.344} C_DIS
LIN {X -0.234,Y -487.204,Z 413.499,A 0.000,B 0.000,C 90.000,E1 269.885} C_DIS
LIN {X 0.105,Y -486.039,Z 413.498,A 0.000,B 0.000,C 90.000,E1 269.599} C_DIS
LIN {X -0.199,Y -483.106,Z 413.495,A 0.000,B 0.000,C 90.000,E1 269.141} C_DIS
LIN {X -0.038,Y -479.351,Z 413.492,A 0.000,B 0.000,C 90.000,E1 268.625} C_DIS
LIN {X 0.115,Y -474.585,Z 413.490,A 0.000,B 0.000,C 90.000,E1 268.108} C_DIS
LIN {X -0.047,Y -468.884,Z 413.487,A 0.000,B 0.000,C 90.000,E1 267.650} C_DIS
LIN {X -0.193,Y -462.394,Z 413.485,A 0.000,B 0.000,C 90.000,E1 267.249} C_DIS
LIN {X -0.229,Y -455.437,Z 413.483,A 0.000,B 0.000,C 90.000,E1 266.906} C_DIS
LIN {X -0.178,Y -448.242,Z 413.481,A 0.000,B 0.000,C 90.000,E1 266.617} C_DIS
LIN {X -0.174,Y -441.020,Z 413.480,A 0.000,B 0.000,C 90.000,E1 266.388} C_DIS
LIN {X 0.187,Y -433.286,Z 413.479,A 0.000,B 0.000,C 90.000,E1 266.159} C_DIS
LIN {X 0.035,Y -424.632,Z 413.478,A 0.000,B 0.000,C 90.000,E1 266.045} C_DIS
LIN {X 0.185,Y -412.461,Z 413.478,A 0.000,B 0.000,C 90.000,E1 265.931} C_DIS
LIN {X 0.145,Y -409.446,Z 413.477,A 0.000,B 0.000,C 90.000,E1 265.927} C_DIS
LIN {X 0.034,Y -180.918,Z 413.477,A 0.000,B 0.000,C 90.000,E1 265.927} C_DIS
LIN {X 0.037,Y -180.837,Z 413.472,A 0.000,B 0.000,C 90.000,E1 264.894} C_DIS
LIN {X -0.066,Y -178.878,Z 413.443,A 0.000,B 0.000,C 90.000,E1 259.690} C_DIS
LIN {X 0.011,Y -175.921,Z 413.414,A 0.000,B 0.000,C 90.000,E1 254.574} C_DIS
LIN {X -0.100,Y -174.618,Z 413.405,A 0.000,B 0.000,C 90.000,E1 252.906} C_DIS
LIN {X -0.007,Y -171.599,Z 413.381,A 0.000,B 0.000,C 90.000,E1 248.592} C_DIS
LIN {X -0.018,Y -167.821,Z 413.357,A 0.000,B 0.000,C 90.000,E1 244.280} C_DIS
LIN {X -0.002,Y -166.545,Z 413.347,A 0.000,B 0.000,C 90.000,E1 242.538} C_DIS
LIN {X -0.090,Y -162.541,Z 413.323,A 0.000,B 0.000,C 90.000,E1 238.201} C_DIS
LIN {X -0.030,Y -161.218,Z 413.313,A 0.000,B 0.000,C 90.000,E1 236.421} C_DIS
LIN {X 0.005,Y -157.225,Z 413.289,A 0.000,B 0.000,C 90.000,E1 231.984} C_DIS
LIN {X 0.028,Y -155.951,Z 413.279,A 0.000,B 0.000,C 90.000,E1 230.194} C_DIS
LIN {X -0.013,Y -152.203,Z 413.254,A 0.000,B 0.000,C 90.000,E1 225.729} C_DIS
LIN {X 0.008,Y -150.449,Z 413.239,A 0.000,B 0.000,C 90.000,E1 223.014} C_DIS
LIN {X 0.034,Y -147.175,Z 413.214,A 0.000,B 0.000,C 90.000,E1 218.463} C_DIS
LIN {X 0.001,Y -145.192,Z 413.193,A 0.000,B 0.000,C 90.000,E1 214.818} C_DIS
LIN {X 0.037,Y -142.333,Z 413.163,A 0.000,B 0.000,C 90.000,E1 209.283} C_DIS
LIN {X -0.035,Y -141.722,Z 413.152,A 0.000,B 0.000,C 90.000,E1 207.462} C_DIS
LIN {X -0.052,Y -139.478,Z 413.116,A 0.000,B 0.000,C 90.000,E1 200.972} C_DIS
LIN {X -0.063,Y -138.975,Z 413.101,A 0.000,B 0.000,C 90.000,E1 198.181} C_DIS
LIN {X 0.058,Y -138.331,Z 413.054,A 0.000,B 0.000,C 90.000,E1 189.726} C_DIS
LIN {X 0.061,Y -139.432,Z 413.007,A 0.000,B 0.000,C 90.000,E1 181.318} C_DIS
LIN {X 0.002,Y -140.960,Z 412.976,A 0.000,B 0.000,C 90.000,E1 175.755} C_DIS
LIN {X -0.048,Y -142.715,Z 412.956,A 0.000,B 0.000,C 90.000,E1 172.064} C_DIS
LIN {X 0.051,Y -145.094,Z 412.930,A 0.000,B 0.000,C 90.000,E1 167.409} C_DIS
LIN {X 0.047,Y -147.719,Z 412.910,A 0.000,B 0.000,C 90.000,E1 163.740} C_DIS
LIN {X -0.012,Y -150.376,Z 412.889,A 0.000,B 0.000,C 90.000,E1 160.115} C_DIS
LIN {X 0.005,Y -153.805,Z 412.869,A 0.000,B 0.000,C 90.000,E1 156.485} C_DIS
LIN {X 0.065,Y -157.217,Z 412.849,A 0.000,B 0.000,C 90.000,E1 152.871} C_DIS
LIN {X 0.006,Y -161.383,Z 412.830,A 0.000,B 0.000,C 90.000,E1 149.331} C_DIS
LIN {X 0.017,Y -165.585,Z 412.810,A 0.000,B 0.000,C 90.000,E1 145.801} C_DIS
LIN {X 0.003,Y -170.507,Z 412.791,A 0.000,B 0.000,C 90.000,E1 142.316} C_DIS
LIN {X 0.048,Y -175.386,Z 412.771,A 0.000,B 0.000,C 90.000,E1 138.852} C_DIS
LIN {X -0.090,Y -181.010,Z 412.753,A 0.000,B 0.000,C 90.000,E1 135.486} C_DIS
LIN {X 0.034,Y -186.440,Z 412.734,A 0.000,B 0.000,C 90.000,E1 132.081} C_DIS
LIN {X 0.103,Y -191.065,Z 412.720,A 0.000,B 0.000,C 90.000,E1 129.564} C_DIS
LIN {X 0.017,Y -196.946,Z 412.701,A 0.000,B 0.000,C 90.000,E1 126.251} C_DIS
LIN {X -0.028,Y -295.912,Z 412.701,A 0.000,B 0.000,C 90.000,E1 126.251} C_DIS
LIN {X 0.198,Y -301.367,Z 412.700,A 0.000,B 0.000,C 90.000,E1 126.011} C_DIS
LIN {X -0.119,Y -303.781,Z 412.699,A 0.000,B 0.000,C 90.000,E1 125.884} C_DIS
LIN {X -0.157,Y -307.047,Z 412.697,A 0.000,B 0.000,C 90.000,E1 125.518} C_DIS
LIN {X -0.045,Y -309.010,Z 412.695,A 0.000,B 0.000,C 90.000,E1 125.185} C_DIS
LIN {X -0.007,Y -310.553,Z 412.694,A 0.000,B 0.000,C 90.000,E1 124.865} C_DIS
LIN {X 0.078,Y -312.881,Z 412.690,A 0.000,B 0.000,C 90.000,E1 124.199} C_DIS
LIN {X -0.115,Y -322.789,Z 412.674,A 0.000,B 0.000,C 90.000,E1 121.337} C_DIS
LIN {X -0.092,Y -334.024,Z 412.658,A 0.000,B 0.000,C 90.000,E1 118.487} C_DIS
LIN {X 0.087,Y -346.679,Z 412.643,A 0.000,B 0.000,C 90.000,E1 115.668} C_DIS
LIN {X -0.033,Y -359.220,Z 412.629,A 0.000,B 0.000,C 90.000,E1 113.259} C_DIS
LIN {X 0.069,Y -373.066,Z 412.616,A 0.000,B 0.000,C 90.000,E1 110.865} C_DIS
LIN {X 0.047,Y -388.320,Z 412.603,A 0.000,B 0.000,C 90.000,E1 108.544} C_DIS
LIN {X 0.154,Y -405.096,Z 412.590,A 0.000,B 0.000,C 90.000,E1 106.260} C_DIS
LIN {X 0.061,Y -423.516,Z 412.578,A 0.000,B 0.000,C 90.000,E1 104.064} C_DIS
LIN {X 0.047,Y -443.387,Z 412.566,A 0.000,B 0.000,C 90.000,E1 101.951} C_DIS
LIN {X -0.031,Y -463.880,Z 412.556,A 0.000,B 0.000,C 90.000,E1 100.018} C_DIS
LIN {X 0.222,Y -487.430,Z 412.545,A 0.000,B 0.000,C 90.000,E1 97.992} C_DIS
LIN {X -0.042,Y -490.981,Z 412.542,A 0.000,B 0.000,C 90.000,E1 97.587} C_DIS
LIN {X -0.150,Y -492.318,Z 412.541,A 0.000,B 0.000,C 90.000,E1 97.352} C_DIS
LIN {X 0.169,Y -493.303,Z 412.539,A 0.000,B 0.000,C 90.000,E1 97.068} C_DIS
LIN {X -0.082,Y -494.400,Z 412.537,A 0.000,B 0.000,C 90.000,E1 96.606} C_DIS
LIN {X 0.164,Y -494.483,Z 412.534,A 0.000,B 0.000,C 90.000,E1 96.087} C_DIS
LIN {X -0.077,Y -493.566,Z 412.531,A 0.000,B 0.000,C 90.000,E1 95.625} C_DIS
LIN {X 0.173,Y -491.486,Z 412.528,A 0.000,B 0.000,C 90.000,E1 95.106} C_DIS
LIN {X 0.028,Y -489.870,Z 412.527,A 0.000,B 0.000,C 90.000,E1 94.878} C_DIS
LIN {X -0.020,Y -482.238,Z 412.522,A 0.000,B 0.000,C 90.000,E1 93.898} C_DIS
LIN {X 0.007,Y -466.323,Z 412.511,A 0.000,B 0.000,C 90.000,E1 91.892} C_DIS
LIN {X 0.142,Y -451.306,Z 412.499,A 0.000,B 0.000,C 90.000,E1 89.828} C_DIS
LIN {X 0.168,Y -430.763,Z 412.482,A 0.000,B 0.000,C 90.000,E1 86.674} C_DIS
LIN {X 0.017,Y -411.754,Z 412.464,A 0.000,B 0.000,C 90.000,E1 83.451} C_DIS
LIN {X -0.093,Y -399.472,Z 412.451,A 0.000,B 0.000,C 90.000,E1 81.254} C_DIS
LIN {X -0.050,Y -387.432,Z 412.439,A 0.000,B 0.000,C 90.000,E1 78.993} C_DIS
LIN {X -0.054,Y -372.766,Z 412.423,A 0.000,B 0.000,C 90.000,E1 76.117} C_DIS
LIN {X 0.079,Y -360.014,Z 412.408,A 0.000,B 0.000,C 90.000,E1 73.449} C_DIS
LIN {X 0.104,Y -345.359,Z 412.390,A 0.000,B 0.000,C 90.000,E1 70.134} C_DIS
LIN {X 0.155,Y -333.907,Z 412.374,A 0.000,B 0.000,C 90.000,E1 67.358} C_DIS
LIN {X 0.199,Y -323.962,Z 412.360,A 0.000,B 0.000,C 90.000,E1 64.845} C_DIS
LIN {X -0.083,Y -313.155,Z 412.345,A 0.000,B 0.000,C 90.000,E1 62.025} C_DIS
LIN {X 0.059,Y -302.856,Z 412.328,A 0.000,B 0.000,C 90.000,E1 59.076} C_DIS
LIN {X -0.112,Y -292.234,Z 412.310,A 0.000,B 0.000,C 90.000,E1 55.801} C_DIS
LIN {X 0.074,Y -282.551,Z 412.291,A 0.000,B 0.000,C 90.000,E1 52.396} C_DIS
LIN {X 0.037,Y -275.088,Z 412.276,A 0.000,B 0.000,C 90.000,E1 49.666} C_DIS
LIN {X -0.001,Y -269.322,Z 412.264,A 0.000,B 0.000,C 90.000,E1 47.595} C_DIS
LIN {X 0.033,Y -263.334,Z 412.253,A 0.000,B 0.000,C 90.000,E1 45.486} C_DIS
LIN {X -0.054,Y -257.230,Z 412.241,A 0.000,B 0.000,C 90.000,E1 43.380} C_DIS
LIN {X -0.011,Y -248.845,Z 412.225,A 0.000,B 0.000,C 90.000,E1 40.496} C_DIS
LIN {X 0.009,Y -240.613,Z 412.209,A 0.000,B 0.000,C 90.000,E1 37.569} C_DIS
LIN {X -0.048,Y -232.751,Z 412.192,A 0.000,B 0.000,C 90.000,E1 34.612} C_DIS
LIN {X -0.042,Y -225.593,Z 412.175,A 0.000,B 0.000,C 90.000,E1 31.592} C_DIS
LIN {X 0.122,Y -219.036,Z 412.158,A 0.000,B 0.000,C 90.000,E1 28.487} C_DIS
LIN {X 0.008,Y -213.180,Z 412.141,A 0.000,B 0.000,C 90.000,E1 25.412} C_DIS
LIN {X 0.065,Y -206.759,Z 412.119,A 0.000,B 0.000,C 90.000,E1 21.461} C_DIS
LIN {X -0.072,Y -201.234,Z 412.097,A 0.000,B 0.000,C 90.000,E1 17.511} C_DIS
LIN {X -0.037,Y -196.778,Z 412.075,A 0.000,B 0.000,C 90.000,E1 13.467} C_DIS
LIN {X 0.018,Y -193.206,Z 412.052,A 0.000,B 0.000,C 90.000,E1 9.378} C_DIS
LIN {X -0.060,Y -190.353,Z 412.025,A 0.000,B 0.000,C 90.000,E1 4.473} C_DIS
LIN {X 0.071,Y -189.063,Z 411.993,A 0.000,B 0.000,C 90.000,E1 358.682} C_DIS
LIN {X -0.023,Y -191.021,Z 411.947,A 0.000,B 0.000,C 90.000,E1 350.443} C_DIS
LIN {X -0.059,Y -194.061,Z 411.919,A 0.000,B 0.000,C 90.000,E1 345.519} C_DIS
LIN {X 0.051,Y -197.623,Z 411.897,A 0.000,B 0.000,C 90.000,E1 341.402} C_DIS
LIN {X 0.027,Y -202.262,Z 411.874,A 0.000,B 0.000,C 90.000,E1 337.358} C_DIS
LIN {X -0.094,Y -207.953,Z 411.852,A 0.000,B 0.000,C 90.000,E1 333.384} C_DIS
LIN {X -0.033,Y -214.506,Z 411.830,A 0.000,B 0.000,C 90.000,E1 329.410} C_DIS
LIN {X -0.058,Y -221.704,Z 411.808,A 0.000,B 0.000,C 90.000,E1 325.515} C_DIS
LIN {X -0.037,Y -227.882,Z 411.791,A 0.000,B 0.000,C 90.000,E1 322.431} C_DIS
LIN {X 0.092,Y -236.472,Z 411.770,A 0.000,B 0.000,C 90.000,E1 318.609} C_DIS
LIN {X -0.017,Y -245.310,Z 411.752,A 0.000,B 0.000,C 90.000,E1 315.283} C_DIS
LIN {X 0.119,Y -252.965,Z 411.737,A 0.000,B 0.000,C 90.000,E1 312.690} C_DIS
LIN {X -0.003,Y -264.047,Z 411.719,A 0.000,B 0.000,C 90.000,E1 309.483} C_DIS
LIN {X 0.012,Y -274.685,Z 411.704,A 0.000,B 0.000,C 90.000,E1 306.664} C_DIS
LIN {X 0.063,Y -288.867,Z 411.685,A 0.000,B 0.000,C 90.000,E1 303.214} C_DIS
LIN {X 0.019,Y -303.706,Z 411.666,A 0.000,B 0.000,C 90.000,E1 299.873} C_DIS
LIN {X -0.058,Y -318.686,Z 411.650,A 0.000,B 0.000,C 90.000,E1 296.950} C_DIS
LIN {X 0.043,Y -333.323,Z 411.636,A 0.000,B 0.000,C 90.000,E1 294.387} C_DIS
LIN {X 0.085,Y -345.489,Z 411.625,A 0.000,B 0.000,C 90.000,E1 292.514} C_DIS
LIN {X -0.003,Y -367.522,Z 411.608,A 0.000,B 0.000,C 90.000,E1 289.504} C_DIS
LIN {X -0.003,Y -383.994,Z 411.597,A 0.000,B 0.000,C 90.000,E1 287.457} C_DIS
LIN {X -0.164,Y -404.555,Z 411.585,A 0.000,B 0.000,C 90.000,E1 285.245} C_DIS
LIN {X 0.155,Y -422.643,Z 411.575,A 0.000,B 0.000,C 90.000,E1 283.411} C_DIS
LIN {X -0.033,Y -435.409,Z 411.568,A 0.000,B 0.000,C 90.000,E1 282.175} C_DIS
LIN {X -0.118,Y -442.759,Z 411.563,A 0.000,B 0.000,C 90.000,E1 281.422} C_DIS
LIN {X -0.165,Y -449.585,Z 411.559,A 0.000,B 0.000,C 90.000,E1 280.658} C_DIS
LIN {X -0.004,Y -457.857,Z 411.553,A 0.000,B 0.000,C 90.000,E1 279.613} C_DIS
LIN {X 0.121,Y -465.458,Z 411.548,A 0.000,B 0.000,C 90.000,E1 278.568} C_DIS
LIN {X -0.196,Y -472.338,Z 411.542,A 0.000,B 0.000,C 90.000,E1 277.587} C_DIS
LIN {X 0.039,Y -478.527,Z 411.536,A 0.000,B 0.000,C 90.000,E1 276.549} C_DIS
LIN {X 0.050,Y -482.661,Z 411.532,A 0.000,B 0.000,C 90.000,E1 275.796} C_DIS
LIN {X 0.221,Y -485.018,Z 411.529,A 0.000,B 0.000,C 90.000,E1 275.277} C_DIS
LIN {X -0.119,Y -487.048,Z 411.527,A 0.000,B 0.000,C 90.000,E1 274.821} C_DIS
LIN {X 0.074,Y -488.732,Z 411.524,A 0.000,B 0.000,C 90.000,E1 274.302} C_DIS
LIN {X -0.212,Y -490.042,Z 411.521,A 0.000,B 0.000,C 90.000,E1 273.841} C_DIS
LIN {X -0.032,Y -491.015,Z 411.518,A 0.000,B 0.000,C 90.000,E1 273.326} C_DIS
LIN {X 0.185,Y -491.669,Z 411.516,A 0.000,B 0.000,C 90.000,E1 272.808} C_DIS
LIN {X -0.108,Y -491.998,Z 411.513,A 0.000,B 0.000,C 90.000,E1 272.350} C_DIS
LIN {X 0.097,Y -491.890,Z 411.510,A 0.000,B 0.000,C 90.000,E1 271.835} C_DIS
LIN {X -0.174,Y -491.475,Z 411.508,A 0.000,B 0.000,C 90.000,E1 271.375} C_DIS
LIN {X 0.031,Y -490.565,Z 411.505,A 0.000,B 0.000,C 90.000,E1 270.859} C_DIS
LIN {X 0.235,Y -489.230,Z 411.502,A 0.000,B 0.000,C 90.000,E1 270.344} C_DIS
LIN {X -0.055,Y -487.321,Z 411.499,A 0.000,B 0.000,C 90.000,E1 269.885} C_DIS
LIN {X -0.203,Y -486.164,Z 411.498,A 0.000,B 0.000,C 90.000,E1 269.656} C_DIS
LIN {X -0.021,Y -483.296,Z 411.495,A 0.000,B 0.000,C 90.000,E1 269.141} C_DIS
LIN {X 0.139,Y -479.568,Z 411.492,A 0.000,B 0.000,C 90.000,E1 268.625} C_DIS
LIN {X -0.024,Y -477.385,Z 411.491,A 0.000,B 0.000,C 90.000,E1 268.396} C_DIS
LIN {X 0.120,Y -472.098,Z 411.488,A 0.000,B 0.000,C 90.000,E1 267.879} C_DIS
LIN {X 0.103,Y -469.194,Z 411.487,A 0.000,B 0.000,C 90.000,E1 267.650} C_DIS
LIN {X -0.074,Y -462.701,Z 411.485,A 0.000,B 0.000,C 90.000,E1 267.249} C_DIS
LIN {X -0.231,Y -459.194,Z 411.484,A 0.000,B 0.000,C 90.000,E1 267.078} C_DIS
LIN {X -0.018,Y -451.921,Z 411.482,A 0.000,B 0.000,C 90.000,E1 266.731} C_DIS
LIN {X -0.214,Y -444.742,Z 411.480,A 0.000,B 0.000,C 90.000,E1 266.502} C_DIS
LIN {X -0.047,Y -437.206,Z 411.479,A 0.000,B 0.000,C 90.000,E1 266.274} C_DIS
LIN {X 0.036,Y -428.924,Z 411.478,A 0.000,B 0.000,C 90.000,E1 266.102} C_DIS
LIN {X 0.044,Y -418.965,Z 411.478,A 0.000,B 0.000,C 90.000,E1 265.988} C_DIS
LIN {X 0.142,Y -409.026,Z 411.477,A 0.000,B 0.000,C 90.000,E1 265.927} C_DIS
LIN {X 0.033,Y -180.918,Z 411.477,A 0.000,B 0.000,C 90.000,E1 265.927} C_DIS
LIN {X 0.036,Y -180.837,Z 411.472,A 0.000,B 0.000,C 90.000,E1 264.894} C_DIS
LIN {X -0.067,Y -178.878,Z 411.443,A 0.000,B 0.000,C 90.000,E1 259.690} C_DIS
LIN {X 0.009,Y -175.920,Z 411.414,A 0.000,B 0.000,C 90.000,E1 254.574} C_DIS
LIN {X 0.065,Y -174.617,Z 411.405,A 0.000,B 0.000,C 90.000,E1 252.851} C_DIS
LIN {X -0.009,Y -171.598,Z 411.381,A 0.000,B 0.000,C 90.000,E1 248.592} C_DIS
LIN {X -0.020,Y -167.821,Z 411.357,A 0.000,B 0.000,C 90.000,E1 244.280} C_DIS
LIN {X -0.002,Y -166.544,Z 411.347,A 0.000,B 0.000,C 90.000,E1 242.538} C_DIS
LIN {X -0.091,Y -162.541,Z 411.323,A 0.000,B 0.000,C 90.000,E1 238.201} C_DIS
LIN {X -0.032,Y -161.217,Z 411.313,A 0.000,B 0.000,C 90.000,E1 236.421} C_DIS
LIN {X 0.004,Y -157.225,Z 411.289,A 0.000,B 0.000,C 90.000,E1 231.984} C_DIS
LIN {X 0.027,Y -155.950,Z 411.279,A 0.000,B 0.000,C 90.000,E1 230.194} C_DIS
LIN {X -0.015,Y -152.203,Z 411.254,A 0.000,B 0.000,C 90.000,E1 225.729} C_DIS
LIN {X 0.006,Y -150.449,Z 411.239,A 0.000,B 0.000,C 90.000,E1 223.014} C_DIS
LIN {X 0.034,Y -147.174,Z 411.214,A 0.000,B 0.000,C 90.000,E1 218.463} C_DIS
LIN {X 0.000,Y -145.191,Z 411.193,A 0.000,B 0.000,C 90.000,E1 214.818} C_DIS
LIN {X 0.035,Y -142.333,Z 411.163,A 0.000,B 0.000,C 90.000,E1 209.283} C_DIS
LIN {X -0.036,Y -141.721,Z 411.152,A 0.000,B 0.000,C 90.000,E1 207.462} C_DIS
LIN {X -0.053,Y -139.477,Z 411.116,A 0.000,B 0.000,C 90.000,E1 200.972} C_DIS
LIN {X -0.064,Y -138.975,Z 411.101,A 0.000,B 0.000,C 90.000,E1 198.181} C_DIS
LIN {X 0.057,Y -138.331,Z 411.054,A 0.000,B 0.000,C 90.000,E1 189.726} C_DIS
LIN {X 0.060,Y -139.432,Z 411.007,A 0.000,B 0.000,C 90.000,E1 181.318} C_DIS
LIN {X 0.001,Y -140.960,Z 410.976,A 0.000,B 0.000,C 90.000,E1 175.755} C_DIS
LIN {X -0.049,Y -142.715,Z 410.956,A 0.000,B 0.000,C 90.000,E1 172.064} C_DIS
LIN {X 0.050,Y -145.094,Z 410.930,A 0.000,B 0.000,C 90.000,E1 167.409} C_DIS
LIN {X 0.045,Y -147.718,Z 410.910,A 0.000,B 0.000,C 90.000,E1 163.740} C_DIS
LIN {X -0.013,Y -150.377,Z 410.889,A 0.000,B 0.000,C 90.000,E1 160.115} C_DIS
LIN {X 0.004,Y -153.806,Z 410.869,A 0.000,B 0.000,C 90.000,E1 156.485} C_DIS
LIN {X 0.064,Y -157.217,Z 410.849,A 0.000,B 0.000,C 90.000,E1 152.871} C_DIS
LIN {X 0.005,Y -161.384,Z 410.830,A 0.000,B 0.000,C 90.000,E1 149.331} C_DIS
LIN {X 0.016,Y -165.586,Z 410.810,A 0.000,B 0.000,C 90.000,E1 145.801} C_DIS
LIN {X 0.002,Y -170.507,Z 410.791,A 0.000,B 0.000,C 90.000,E1 142.316} C_DIS
LIN {X 0.047,Y -175.387,Z 410.771,A 0.000,B 0.000,C 90.000,E1 138.852} C_DIS
LIN {X -0.091,Y -181.011,Z 410.753,A 0.000,B 0.000,C 90.000,E1 135.486} C_DIS
LIN {X 0.033,Y -186.441,Z 410.734,A 0.000,B 0.000,C 90.000,E1 132.081} C_DIS
LIN {X 0.102,Y -191.066,Z 410.720,A 0.000,B 0.000,C 90.000,E1 129.564} C_DIS
LIN {X -0.070,Y -197.059,Z 410.701,A 0.000,B 0.000,C 90.000,E1 126.217} C_DIS
LIN {X 0.081,Y -296.330,Z 410.701,A 0.000,B 0.000,C 90.000,E1 126.171} C_DIS
LIN {X -0.024,Y -297.485,Z 410.701,A 0.000,B 0.000,C 90.000,E1 126.171} C_DIS
LIN {X -0.073,Y -301.454,Z 410.700,A 0.000,B 0.000,C 90.000,E1 126.011} C_DIS
LIN {X 0.122,Y -303.700,Z 410.699,A 0.000,B 0.000,C 90.000,E1 125.804} C_DIS
LIN {X -0.159,Y -306.798,Z 410.697,A 0.000,B 0.000,C 90.000,E1 125.518} C_DIS
LIN {X 0.006,Y -308.799,Z 410.695,A 0.000,B 0.000,C 90.000,E1 125.185} C_DIS
LIN {X -0.081,Y -310.372,Z 410.694,A 0.000,B 0.000,C 90.000,E1 124.898} C_DIS
LIN {X 0.138,Y -311.719,Z 410.692,A 0.000,B 0.000,C 90.000,E1 124.532} C_DIS
LIN {X 0.073,Y -323.882,Z 410.672,A 0.000,B 0.000,C 90.000,E1 121.003} C_DIS
LIN {X -0.022,Y -335.257,Z 410.657,A 0.000,B 0.000,C 90.000,E1 118.180} C_DIS
LIN {X -0.113,Y -348.072,Z 410.641,A 0.000,B 0.000,C 90.000,E1 115.412} C_DIS
LIN {X 0.123,Y -360.761,Z 410.628,A 0.000,B 0.000,C 90.000,E1 112.950} C_DIS
LIN {X -0.078,Y -374.768,Z 410.614,A 0.000,B 0.000,C 90.000,E1 110.610} C_DIS
LIN {X -0.072,Y -390.196,Z 410.602,A 0.000,B 0.000,C 90.000,E1 108.290} C_DIS
LIN {X -0.046,Y -407.159,Z 410.589,A 0.000,B 0.000,C 90.000,E1 106.024} C_DIS
LIN {X -0.097,Y -425.783,Z 410.577,A 0.000,B 0.000,C 90.000,E1 103.828} C_DIS
LIN {X 0.020,Y -445.764,Z 410.565,A 0.000,B 0.000,C 90.000,E1 101.715} C_DIS
LIN {X 0.016,Y -466.319,Z 410.554,A 0.000,B 0.000,C 90.000,E1 99.792} C_DIS
LIN {X -0.164,Y -487.305,Z 410.545,A 0.000,B 0.000,C 90.000,E1 98.049} C_DIS
LIN {X 0.103,Y -490.950,Z 410.542,A 0.000,B 0.000,C 90.000,E1 97.587} C_DIS
LIN {X -0.006,Y -492.341,Z 410.541,A 0.000,B 0.000,C 90.000,E1 97.352} C_DIS
LIN {X -0.177,Y -493.373,Z 410.539,A 0.000,B 0.000,C 90.000,E1 97.125} C_DIS
LIN {X 0.063,Y -494.546,Z 410.537,A 0.000,B 0.000,C 90.000,E1 96.606} C_DIS
LIN {X -0.183,Y -494.698,Z 410.534,A 0.000,B 0.000,C 90.000,E1 96.144} C_DIS
LIN {X 0.069,Y -493.853,Z 410.531,A 0.000,B 0.000,C 90.000,E1 95.625} C_DIS
LIN {X -0.171,Y -491.862,Z 410.529,A 0.000,B 0.000,C 90.000,E1 95.163} C_DIS
LIN {X 0.174,Y -490.310,Z 410.527,A 0.000,B 0.000,C 90.000,E1 94.878} C_DIS
LIN {X 0.128,Y -482.708,Z 410.522,A 0.000,B 0.000,C 90.000,E1 93.898} C_DIS
LIN {X -0.112,Y -468.754,Z 410.512,A 0.000,B 0.000,C 90.000,E1 92.178} C_DIS
LIN {X -0.150,Y -451.745,Z 410.499,A 0.000,B 0.000,C 90.000,E1 89.885} C_DIS
LIN {X 0.053,Y -429.502,Z 410.480,A 0.000,B 0.000,C 90.000,E1 86.445} C_DIS
LIN {X -0.143,Y -410.578,Z 410.462,A 0.000,B 0.000,C 90.000,E1 83.223} C_DIS
LIN {X 0.109,Y -398.311,Z 410.450,A 0.000,B 0.000,C 90.000,E1 80.971} C_DIS
LIN {X -0.199,Y -386.305,Z 410.437,A 0.000,B 0.000,C 90.000,E1 78.757} C_DIS
LIN {X 0.132,Y -371.690,Z 410.421,A 0.000,B 0.000,C 90.000,E1 75.825} C_DIS
LIN {X -0.021,Y -358.978,Z 410.407,A 0.000,B 0.000,C 90.000,E1 73.196} C_DIS
LIN {X -0.008,Y -344.355,Z 410.388,A 0.000,B 0.000,C 90.000,E1 69.880} C_DIS
LIN {X 0.022,Y -332.858,Z 410.373,A 0.000,B 0.000,C 90.000,E1 67.102} C_DIS
LIN {X 0.000,Y -321.679,Z 410.357,A 0.000,B 0.000,C 90.000,E1 64.280} C_DIS
LIN {X 0.136,Y -309.847,Z 410.339,A 0.000,B 0.000,C 90.000,E1 61.051} C_DIS
LIN {X 0.090,Y -298.624,Z 410.321,A 0.000,B 0.000,C 90.000,E1 57.788} C_DIS
LIN {X -0.032,Y -288.417,Z 410.303,A 0.000,B 0.000,C 90.000,E1 54.482} C_DIS
LIN {X -0.025,Y -278.917,Z 410.284,A 0.000,B 0.000,C 90.000,E1 51.090} C_DIS
LIN {X 0.035,Y -273.333,Z 410.272,A 0.000,B 0.000,C 90.000,E1 49.013} C_DIS
LIN {X -0.043,Y -267.500,Z 410.261,A 0.000,B 0.000,C 90.000,E1 46.944} C_DIS
LIN {X -0.054,Y -261.499,Z 410.249,A 0.000,B 0.000,C 90.000,E1 44.838} C_DIS
LIN {X 0.012,Y -255.316,Z 410.237,A 0.000,B 0.000,C 90.000,E1 42.690} C_DIS
LIN {X -0.026,Y -249.077,Z 410.225,A 0.000,B 0.000,C 90.000,E1 40.539} C_DIS
LIN {X 0.037,Y -240.854,Z 410.209,A 0.000,B 0.000,C 90.000,E1 37.604} C_DIS
LIN {X 0.127,Y -233.001,Z 410.192,A 0.000,B 0.000,C 90.000,E1 34.612} C_DIS
LIN {X 0.014,Y -225.839,Z 410.176,A 0.000,B 0.000,C 90.000,E1 31.623} C_DIS
LIN {X 0.000,Y -219.254,Z 410.159,A 0.000,B 0.000,C 90.000,E1 28.565} C_DIS
LIN {X -0.008,Y -213.335,Z 410.141,A 0.000,B 0.000,C 90.000,E1 25.463} C_DIS
LIN {X -0.027,Y -206.877,Z 410.120,A 0.000,B 0.000,C 90.000,E1 21.535} C_DIS
LIN {X 0.103,Y -201.306,Z 410.097,A 0.000,B 0.000,C 90.000,E1 17.511} C_DIS
LIN {X -0.102,Y -196.791,Z 410.075,A 0.000,B 0.000,C 90.000,E1 13.536} C_DIS
LIN {X -0.035,Y -193.182,Z 410.052,A 0.000,B 0.000,C 90.000,E1 9.443} C_DIS
LIN {X -0.084,Y -190.309,Z 410.025,A 0.000,B 0.000,C 90.000,E1 4.531} C_DIS
LIN {X 0.070,Y -188.970,Z 409.993,A 0.000,B 0.000,C 90.000,E1 358.682} C_DIS
LIN {X -0.030,Y -190.903,Z 409.947,A 0.000,B 0.000,C 90.000,E1 350.443} C_DIS
LIN {X -0.071,Y -193.925,Z 409.919,A 0.000,B 0.000,C 90.000,E1 345.519} C_DIS
LIN {X 0.034,Y -197.466,Z 409.897,A 0.000,B 0.000,C 90.000,E1 341.402} C_DIS
LIN {X 0.005,Y -202.118,Z 409.874,A 0.000,B 0.000,C 90.000,E1 337.358} C_DIS
LIN {X 0.064,Y -207.798,Z 409.852,A 0.000,B 0.000,C 90.000,E1 333.332} C_DIS
LIN {X -0.065,Y -214.369,Z 409.830,A 0.000,B 0.000,C 90.000,E1 329.410} C_DIS
LIN {X -0.109,Y -220.099,Z 409.813,A 0.000,B 0.000,C 90.000,E1 326.294} C_DIS
LIN {X 0.060,Y -227.743,Z 409.791,A 0.000,B 0.000,C 90.000,E1 322.396} C_DIS
LIN {X 0.043,Y -236.357,Z 409.770,A 0.000,B 0.000,C 90.000,E1 318.609} C_DIS
LIN {X 0.106,Y -245.201,Z 409.751,A 0.000,B 0.000,C 90.000,E1 315.243} C_DIS
LIN {X 0.068,Y -252.872,Z 409.737,A 0.000,B 0.000,C 90.000,E1 312.690} C_DIS
LIN {X -0.058,Y -263.977,Z 409.719,A 0.000,B 0.000,C 90.000,E1 309.483} C_DIS
LIN {X 0.030,Y -273.260,Z 409.706,A 0.000,B 0.000,C 90.000,E1 306.996} C_DIS
LIN {X -0.093,Y -285.871,Z 409.688,A 0.000,B 0.000,C 90.000,E1 303.913} C_DIS
LIN {X -0.090,Y -297.527,Z 409.673,A 0.000,B 0.000,C 90.000,E1 301.209} C_DIS
LIN {X 0.020,Y -308.445,Z 409.660,A 0.000,B 0.000,C 90.000,E1 298.871} C_DIS
LIN {X -0.131,Y -325.830,Z 409.642,A 0.000,B 0.000,C 90.000,E1 295.668} C_DIS
LIN {X -0.096,Y -337.317,Z 409.632,A 0.000,B 0.000,C 90.000,E1 293.770} C_DIS
LIN {X 0.069,Y -354.203,Z 409.618,A 0.000,B 0.000,C 90.000,E1 291.280} C_DIS
LIN {X 0.040,Y -374.574,Z 409.603,A 0.000,B 0.000,C 90.000,E1 288.598} C_DIS
LIN {X -0.210,Y -386.430,Z 409.595,A 0.000,B 0.000,C 90.000,E1 287.221} C_DIS
LIN {X -0.054,Y -406.827,Z 409.583,A 0.000,B 0.000,C 90.000,E1 285.009} C_DIS
LIN {X -0.168,Y -424.860,Z 409.573,A 0.000,B 0.000,C 90.000,E1 283.244} C_DIS
LIN {X 0.069,Y -437.537,Z 409.566,A 0.000,B 0.000,C 90.000,E1 281.951} C_DIS
LIN {X -0.047,Y -444.908,Z 409.562,A 0.000,B 0.000,C 90.000,E1 281.186} C_DIS
LIN {X 0.199,Y -451.671,Z 409.558,A 0.000,B 0.000,C 90.000,E1 280.366} C_DIS
LIN {X -0.012,Y -457.881,Z 409.553,A 0.000,B 0.000,C 90.000,E1 279.613} C_DIS
LIN {X 0.113,Y -465.493,Z 409.548,A 0.000,B 0.000,C 90.000,E1 278.568} C_DIS
LIN {X -0.204,Y -472.338,Z 409.542,A 0.000,B 0.000,C 90.000,E1 277.587} C_DIS
LIN {X 0.032,Y -478.534,Z 409.536,A 0.000,B 0.000,C 90.000,E1 276.549} C_DIS
LIN {X 0.043,Y -482.662,Z 409.532,A 0.000,B 0.000,C 90.000,E1 275.796} C_DIS
LIN {X 0.214,Y -485.019,Z 409.529,A 0.000,B 0.000,C 90.000,E1 275.277} C_DIS
LIN {X -0.128,Y -487.037,Z 409.527,A 0.000,B 0.000,C 90.000,E1 274.821} C_DIS
LIN {X 0.067,Y -488.693,Z 409.524,A 0.000,B 0.000,C 90.000,E1 274.302} C_DIS
LIN {X -0.220,Y -489.994,Z 409.521,A 0.000,B 0.000,C 90.000,E1 273.841} C_DIS
LIN {X -0.040,Y -490.959,Z 409.518,A 0.000,B 0.000,C 90.000,E1 273.326} C_DIS
LIN {X 0.178,Y -491.600,Z 409.516,A 0.000,B 0.000,C 90.000,E1 272.808} C_DIS
LIN {X -0.117,Y -491.912,Z 409.513,A 0.000,B 0.000,C 90.000,E1 272.350} C_DIS
LIN {X 0.088,Y -491.868,Z 409.510,A 0.000,B 0.000,C 90.000,E1 271.835} C_DIS
LIN {X -0.184,Y -491.416,Z 409.508,A 0.000,B 0.000,C 90.000,E1 271.375} C_DIS
LIN {X 0.022,Y -490.525,Z 409.505,A 0.000,B 0.000,C 90.000,E1 270.859} C_DIS
LIN {X 0.225,Y -489.178,Z 409.502,A 0.000,B 0.000,C 90.000,E1 270.344} C_DIS
LIN {X -0.065,Y -487.318,Z 409.499,A 0.000,B 0.000,C 90.000,E1 269.885} C_DIS
LIN {X 0.125,Y -484.808,Z 409.497,A 0.000,B 0.000,C 90.000,E1 269.370} C_DIS
LIN {X -0.032,Y -483.309,Z 409.495,A 0.000,B 0.000,C 90.000,E1 269.141} C_DIS
LIN {X 0.129,Y -479.630,Z 409.492,A 0.000,B 0.000,C 90.000,E1 268.625} C_DIS
LIN {X -0.192,Y -474.899,Z 409.490,A 0.000,B 0.000,C 90.000,E1 268.165} C_DIS
LIN {X 0.110,Y -472.117,Z 409.488,A 0.000,B 0.000,C 90.000,E1 267.879} C_DIS
LIN {X 0.096,Y -469.213,Z 409.487,A 0.000,B 0.000,C 90.000,E1 267.650} C_DIS
LIN {X -0.092,Y -462.757,Z 409.485,A 0.000,B 0.000,C 90.000,E1 267.249} C_DIS
LIN {X -0.137,Y -455.773,Z 409.483,A 0.000,B 0.000,C 90.000,E1 266.906} C_DIS
LIN {X -0.100,Y -448.671,Z 409.481,A 0.000,B 0.000,C 90.000,E1 266.617} C_DIS
LIN {X -0.127,Y -441.376,Z 409.480,A 0.000,B 0.000,C 90.000,E1 266.388} C_DIS
LIN {X -0.218,Y -433.700,Z 409.479,A 0.000,B 0.000,C 90.000,E1 266.216} C_DIS
LIN {X 0.046,Y -424.880,Z 409.478,A 0.000,B 0.000,C 90.000,E1 266.045} C_DIS
LIN {X 0.187,Y -412.899,Z 409.478,A 0.000,B 0.000,C 90.000,E1 265.931} C_DIS
LIN {X 0.146,Y -409.364,Z 409.477,A 0.000,B 0.000,C 90.000,E1 265.927} C_DIS
LIN {X 0.034,Y -180.918,Z 409.477,A 0.000,B 0.000,C 90.000,E1 265.927} C_DIS
LIN {X 0.036,Y -180.837,Z 409.472,A 0.000,B 0.000,C 90.000,E1 264.894} C_DIS
LIN {X -0.067,Y -178.878,Z 409.443,A 0.000,B 0.000,C 90.000,E1 259.690} C_DIS
LIN {X 0.009,Y -175.920,Z 409.414,A 0.000,B 0.000,C 90.000,E1 254.574} C_DIS
LIN {X 0.065,Y -174.617,Z 409.405,A 0.000,B 0.000,C 90.000,E1 252.851} C_DIS
LIN {X -0.009,Y -171.598,Z 409.381,A 0.000,B 0.000,C 90.000,E1 248.592} C_DIS
LIN {X -0.020,Y -167.821,Z 409.357,A 0.000,B 0.000,C 90.000,E1 244.280} C_DIS
LIN {X -0.002,Y -166.544,Z 409.347,A 0.000,B 0.000,C 90.000,E1 242.538} C_DIS
LIN {X -0.091,Y -162.541,Z 409.323,A 0.000,B 0.000,C 90.000,E1 238.201} C_DIS
LIN {X -0.032,Y -161.217,Z 409.313,A 0.000,B 0.000,C 90.000,E1 236.421} C_DIS
LIN {X 0.004,Y -157.225,Z 409.289,A 0.000,B 0.000,C 90.000,E1 231.984} C_DIS
LIN {X 0.027,Y -155.950,Z 409.279,A 0.000,B 0.000,C 90.000,E1 230.194} C_DIS
LIN {X -0.014,Y -152.203,Z 409.254,A 0.000,B 0.000,C 90.000,E1 225.729} C_DIS
LIN {X 0.007,Y -150.448,Z 409.239,A 0.000,B 0.000,C 90.000,E1 223.014} C_DIS
LIN {X 0.034,Y -147.174,Z 409.214,A 0.000,B 0.000,C 90.000,E1 218.463} C_DIS
LIN {X 0.000,Y -145.191,Z 409.193,A 0.000,B 0.000,C 90.000,E1 214.818} C_DIS
LIN {X 0.035,Y -142.333,Z 409.163,A 0.000,B 0.000,C 90.000,E1 209.283} C_DIS
LIN {X -0.036,Y -141.721,Z 409.152,A 0.000,B 0.000,C 90.000,E1 207.462} C_DIS
LIN {X -0.053,Y -139.477,Z 409.116,A 0.000,B 0.000,C 90.000,E1 200.972} C_DIS
LIN {X -0.064,Y -138.975,Z 409.101,A 0.000,B 0.000,C 90.000,E1 198.181} C_DIS
LIN {X 0.057,Y -138.331,Z 409.054,A 0.000,B 0.000,C 90.000,E1 189.726} C_DIS
LIN {X 0.060,Y -139.432,Z 409.007,A 0.000,B 0.000,C 90.000,E1 181.318} C_DIS
LIN {X 0.001,Y -140.960,Z 408.976,A 0.000,B 0.000,C 90.000,E1 175.755} C_DIS
LIN {X -0.049,Y -142.715,Z 408.956,A 0.000,B 0.000,C 90.000,E1 172.064} C_DIS
LIN {X 0.050,Y -145.094,Z 408.930,A 0.000,B 0.000,C 90.000,E1 167.409} C_DIS
LIN {X 0.046,Y -147.718,Z 408.910,A 0.000,B 0.000,C 90.000,E1 163.740} C_DIS
LIN {X -0.013,Y -150.377,Z 408.889,A 0.000,B 0.000,C 90.000,E1 160.115} C_DIS
LIN {X 0.004,Y -153.806,Z 408.869,A 0.000,B 0.000,C 90.000,E1 156.485} C_DIS
LIN {X 0.064,Y -157.217,Z 408.849,A 0.000,B 0.000,C 90.000,E1 152.871} C_DIS
LIN {X 0.005,Y -161.384,Z 408.830,A 0.000,B 0.000,C 90.000,E1 149.331} C_DIS
LIN {X 0.016,Y -165.586,Z 408.810,A 0.000,B 0.000,C 90.000,E1 145.801} C_DIS
LIN {X 0.002,Y -170.507,Z 408.791,A 0.000,B 0.000,C 90.000,E1 142.316} C_DIS
LIN {X 0.047,Y -175.387,Z 408.771,A 0.000,B 0.000,C 90.000,E1 138.852} C_DIS
LIN {X -0.091,Y -181.011,Z 408.753,A 0.000,B 0.000,C 90.000,E1 135.486} C_DIS
LIN {X 0.033,Y -186.441,Z 408.734,A 0.000,B 0.000,C 90.000,E1 132.081} C_DIS
LIN {X 0.102,Y -191.066,Z 408.720,A 0.000,B 0.000,C 90.000,E1 129.564} C_DIS
LIN {X 0.029,Y -197.158,Z 408.701,A 0.000,B 0.000,C 90.000,E1 126.137} C_DIS
LIN {X 0.009,Y -295.649,Z 408.701,A 0.000,B 0.000,C 90.000,E1 126.137} C_DIS
LIN {X 0.044,Y -298.118,Z 408.701,A 0.000,B 0.000,C 90.000,E1 126.091} C_DIS
LIN {X -0.055,Y -303.605,Z 408.699,A 0.000,B 0.000,C 90.000,E1 125.804} C_DIS
LIN {X -0.159,Y -306.524,Z 408.697,A 0.000,B 0.000,C 90.000,E1 125.518} C_DIS
LIN {X 0.059,Y -308.563,Z 408.696,A 0.000,B 0.000,C 90.000,E1 125.185} C_DIS
LIN {X 0.026,Y -310.169,Z 408.694,A 0.000,B 0.000,C 90.000,E1 124.898} C_DIS
LIN {X -0.188,Y -311.591,Z 408.692,A 0.000,B 0.000,C 90.000,E1 124.612} C_DIS
LIN {X -0.097,Y -323.790,Z 408.672,A 0.000,B 0.000,C 90.000,E1 121.052} C_DIS
LIN {X 0.087,Y -335.156,Z 408.657,A 0.000,B 0.000,C 90.000,E1 118.180} C_DIS
LIN {X -0.003,Y -347.959,Z 408.641,A 0.000,B 0.000,C 90.000,E1 115.412} C_DIS
LIN {X -0.097,Y -360.639,Z 408.628,A 0.000,B 0.000,C 90.000,E1 113.003} C_DIS
LIN {X 0.034,Y -374.636,Z 408.615,A 0.000,B 0.000,C 90.000,E1 110.610} C_DIS
LIN {X -0.082,Y -390.053,Z 408.602,A 0.000,B 0.000,C 90.000,E1 108.308} C_DIS
LIN {X 0.069,Y -407.004,Z 408.589,A 0.000,B 0.000,C 90.000,E1 106.024} C_DIS
LIN {X 0.020,Y -425.615,Z 408.577,A 0.000,B 0.000,C 90.000,E1 103.828} C_DIS
LIN {X 0.131,Y -445.589,Z 408.565,A 0.000,B 0.000,C 90.000,E1 101.715} C_DIS
LIN {X 0.123,Y -466.142,Z 408.554,A 0.000,B 0.000,C 90.000,E1 99.792} C_DIS
LIN {X -0.062,Y -487.161,Z 408.545,A 0.000,B 0.000,C 90.000,E1 98.049} C_DIS
LIN {X -0.249,Y -490.920,Z 408.542,A 0.000,B 0.000,C 90.000,E1 97.644} C_DIS
LIN {X 0.130,Y -492.367,Z 408.541,A 0.000,B 0.000,C 90.000,E1 97.352} C_DIS
LIN {X -0.041,Y -493.442,Z 408.540,A 0.000,B 0.000,C 90.000,E1 97.125} C_DIS
LIN {X 0.199,Y -494.688,Z 408.537,A 0.000,B 0.000,C 90.000,E1 96.606} C_DIS
LIN {X -0.047,Y -494.906,Z 408.534,A 0.000,B 0.000,C 90.000,E1 96.144} C_DIS
LIN {X 0.206,Y -494.130,Z 408.531,A 0.000,B 0.000,C 90.000,E1 95.625} C_DIS
LIN {X -0.034,Y -492.224,Z 408.529,A 0.000,B 0.000,C 90.000,E1 95.163} C_DIS
LIN {X -0.176,Y -490.729,Z 408.527,A 0.000,B 0.000,C 90.000,E1 94.935} C_DIS
LIN {X -0.212,Y -483.169,Z 408.522,A 0.000,B 0.000,C 90.000,E1 93.955} C_DIS
LIN {X 0.217,Y -471.192,Z 408.514,A 0.000,B 0.000,C 90.000,E1 92.407} C_DIS
LIN {X -0.222,Y -453.993,Z 408.501,A 0.000,B 0.000,C 90.000,E1 90.172} C_DIS
LIN {X -0.112,Y -433.184,Z 408.483,A 0.000,B 0.000,C 90.000,E1 87.020} C_DIS
LIN {X 0.006,Y -417.083,Z 408.468,A 0.000,B 0.000,C 90.000,E1 84.318} C_DIS
LIN {X -0.093,Y -406.302,Z 408.458,A 0.000,B 0.000,C 90.000,E1 82.413} C_DIS
LIN {X 0.192,Y -392.638,Z 408.444,A 0.000,B 0.000,C 90.000,E1 79.859} C_DIS
LIN {X 0.131,Y -380.739,Z 408.431,A 0.000,B 0.000,C 90.000,E1 77.589} C_DIS
LIN {X 0.022,Y -367.767,Z 408.417,A 0.000,B 0.000,C 90.000,E1 74.991} C_DIS
LIN {X 0.162,Y -353.844,Z 408.400,A 0.000,B 0.000,C 90.000,E1 72.000} C_DIS
LIN {X 0.208,Y -342.024,Z 408.385,A 0.000,B 0.000,C 90.000,E1 69.263} C_DIS
LIN {X 0.190,Y -331.803,Z 408.371,A 0.000,B 0.000,C 90.000,E1 66.794} C_DIS
LIN {X -0.163,Y -320.631,Z 408.356,A 0.000,B 0.000,C 90.000,E1 64.024} C_DIS
LIN {X -0.106,Y -309.990,Z 408.340,A 0.000,B 0.000,C 90.000,E1 61.129} C_DIS
LIN {X -0.144,Y -298.764,Z 408.321,A 0.000,B 0.000,C 90.000,E1 57.867} C_DIS
LIN {X 0.144,Y -288.537,Z 408.303,A 0.000,B 0.000,C 90.000,E1 54.482} C_DIS
LIN {X 0.149,Y -279.046,Z 408.284,A 0.000,B 0.000,C 90.000,E1 51.090} C_DIS
LIN {X 0.000,Y -273.464,Z 408.273,A 0.000,B 0.000,C 90.000,E1 49.057} C_DIS
LIN {X -0.067,Y -267.650,Z 408.261,A 0.000,B 0.000,C 90.000,E1 46.986} C_DIS
LIN {X 0.117,Y -261.664,Z 408.249,A 0.000,B 0.000,C 90.000,E1 44.838} C_DIS
LIN {X -0.007,Y -255.530,Z 408.237,A 0.000,B 0.000,C 90.000,E1 42.732} C_DIS
LIN {X 0.143,Y -249.305,Z 408.225,A 0.000,B 0.000,C 90.000,E1 40.539} C_DIS
LIN {X 0.015,Y -241.101,Z 408.209,A 0.000,B 0.000,C 90.000,E1 37.649} C_DIS
LIN {X -0.027,Y -233.247,Z 408.193,A 0.000,B 0.000,C 90.000,E1 34.692} C_DIS
LIN {X -0.007,Y -226.082,Z 408.176,A 0.000,B 0.000,C 90.000,E1 31.671} C_DIS
LIN {X -0.033,Y -217.896,Z 408.155,A 0.000,B 0.000,C 90.000,E1 27.847} C_DIS
LIN {X 0.024,Y -212.127,Z 408.137,A 0.000,B 0.000,C 90.000,E1 24.719} C_DIS
LIN {X -0.031,Y -205.800,Z 408.115,A 0.000,B 0.000,C 90.000,E1 20.791} C_DIS
LIN {X 0.020,Y -201.373,Z 408.098,A 0.000,B 0.000,C 90.000,E1 17.583} C_DIS
LIN {X 0.067,Y -196.810,Z 408.075,A 0.000,B 0.000,C 90.000,E1 13.536} C_DIS
LIN {X -0.060,Y -193.158,Z 408.053,A 0.000,B 0.000,C 90.000,E1 9.500} C_DIS
LIN {X 0.078,Y -190.265,Z 408.025,A 0.000,B 0.000,C 90.000,E1 4.531} C_DIS
LIN {X -0.010,Y -188.857,Z 407.988,A 0.000,B 0.000,C 90.000,E1 357.879} C_DIS
LIN {X -0.037,Y -190.787,Z 407.947,A 0.000,B 0.000,C 90.000,E1 350.443} C_DIS
LIN {X -0.082,Y -193.772,Z 407.919,A 0.000,B 0.000,C 90.000,E1 345.519} C_DIS
LIN {X 0.017,Y -197.316,Z 407.897,A 0.000,B 0.000,C 90.000,E1 341.402} C_DIS
LIN {X -0.016,Y -201.974,Z 407.874,A 0.000,B 0.000,C 90.000,E1 337.358} C_DIS
LIN {X -0.041,Y -206.416,Z 407.856,A 0.000,B 0.000,C 90.000,E1 334.152} C_DIS
LIN {X -0.128,Y -212.857,Z 407.834,A 0.000,B 0.000,C 90.000,E1 330.205} C_DIS
LIN {X -0.145,Y -219.969,Z 407.813,A 0.000,B 0.000,C 90.000,E1 326.294} C_DIS
LIN {X 0.018,Y -227.627,Z 407.791,A 0.000,B 0.000,C 90.000,E1 322.396} C_DIS
LIN {X -0.003,Y -236.245,Z 407.770,A 0.000,B 0.000,C 90.000,E1 318.609} C_DIS
LIN {X 0.047,Y -245.093,Z 407.751,A 0.000,B 0.000,C 90.000,E1 315.243} C_DIS
LIN {X 0.021,Y -253.960,Z 407.735,A 0.000,B 0.000,C 90.000,E1 312.324} C_DIS
LIN {X -0.075,Y -265.218,Z 407.717,A 0.000,B 0.000,C 90.000,E1 309.116} C_DIS
LIN {X -0.121,Y -274.543,Z 407.704,A 0.000,B 0.000,C 90.000,E1 306.664} C_DIS
LIN {X -0.081,Y -288.686,Z 407.684,A 0.000,B 0.000,C 90.000,E1 303.214} C_DIS
LIN {X -0.138,Y -303.559,Z 407.666,A 0.000,B 0.000,C 90.000,E1 299.873} C_DIS
LIN {X -0.049,Y -315.154,Z 407.653,A 0.000,B 0.000,C 90.000,E1 297.564} C_DIS
LIN {X -0.092,Y -331.475,Z 407.637,A 0.000,B 0.000,C 90.000,E1 294.695} C_DIS
LIN {X -0.096,Y -345.650,Z 407.625,A 0.000,B 0.000,C 90.000,E1 292.514} C_DIS
LIN {X 0.092,Y -365.526,Z 407.610,A 0.000,B 0.000,C 90.000,E1 289.758} C_DIS
LIN {X 0.023,Y -379.497,Z 407.600,A 0.000,B 0.000,C 90.000,E1 288.000} C_DIS
LIN {X -0.152,Y -402.485,Z 407.586,A 0.000,B 0.000,C 90.000,E1 285.481} C_DIS
LIN {X -0.045,Y -423.103,Z 407.574,A 0.000,B 0.000,C 90.000,E1 283.411} C_DIS
LIN {X 0.149,Y -435.835,Z 407.567,A 0.000,B 0.000,C 90.000,E1 282.119} C_DIS
LIN {X 0.041,Y -443.172,Z 407.563,A 0.000,B 0.000,C 90.000,E1 281.366} C_DIS
LIN {X -0.159,Y -450.146,Z 407.559,A 0.000,B 0.000,C 90.000,E1 280.602} C_DIS
END
